C03639=1023.462,361.874,355.874,171.924,48.820,159.677
C03640=1023.470,362.121,355.836,171.932,48.821,159.679
C03641=1023.477,362.367,355.796,171.939,48.821,159.680
C03642=1023.485,362.615,355.758,171.947,48.820,159.681
C03643=1023.494,362.861,355.718,171.955,48.820,159.682
C03644=1023.502,363.108,355.680,171.963,48.820,159.683
C03645=1023.510,363.355,355.640,171.971,48.820,159.684
C03646=1023.517,363.602,355.602,171.978,48.820,159.685
C03647=1023.526,363.848,355.562,171.986,48.819,159.687
C03648=1023.534,364.095,355.523,171.994,48.820,159.688
C03649=1023.542,364.342,355.484,172.001,48.820,159.689
C03650=1023.551,364.589,355.445,172.009,48.819,159.690
C03651=1023.558,364.836,355.405,172.018,48.819,159.691
C03652=1023.567,365.083,355.366,172.025,48.819,159.692
C03653=1023.575,365.330,355.327,172.033,48.820,159.694
C03654=1023.583,365.576,355.288,172.041,48.819,159.695
C03655=1023.591,365.813,355.250,172.049,48.819,159.696
C03656=1023.599,366.049,355.212,172.057,48.819,159.697
C03657=1023.608,366.287,355.175,172.064,48.819,159.698
C03658=1023.615,366.524,355.137,172.072,48.819,159.700
C03659=1023.623,366.761,355.099,172.080,48.819,159.701
C03660=1023.631,366.998,355.060,172.088,48.820,159.702
C03661=1023.639,367.235,355.023,172.095,48.820,159.703
C03662=1023.647,367.471,354.985,172.103,48.819,159.704
C03663=1023.656,367.719,354.945,172.111,48.820,159.705
C03664=1023.664,367.965,354.906,172.119,48.820,159.707
C03665=1023.673,368.212,354.866,172.127,48.819,159.708
C03666=1023.680,368.459,354.826,172.135,48.820,159.709
C03667=1023.689,368.705,354.787,172.144,48.820,159.710
C03668=1023.697,368.952,354.747,172.151,48.820,159.712
C03669=1023.705,369.198,354.707,172.160,48.821,159.713
C03670=1023.713,369.445,354.667,172.168,48.821,159.714
C03671=1023.722,369.693,354.628,172.177,48.821,159.716
C03672=1023.730,369.939,354.587,172.185,48.821,159.717
C03673=1023.739,370.185,354.548,172.192,48.822,159.718
C03674=1023.747,370.432,354.507,172.201,48.822,159.719
C03675=1023.755,370.678,354.468,172.209,48.822,159.721
C03676=1023.764,370.925,354.427,172.218,48.822,159.722
C03677=1023.772,371.172,354.387,172.226,48.823,159.723
C03678=1023.780,371.418,354.347,172.235,48.823,159.725
C03679=1023.789,371.665,354.307,172.243,48.823,159.726
C03680=1023.797,371.912,354.266,172.250,48.824,159.727
C03681=1023.806,372.158,354.226,172.259,48.824,159.729
C03682=1023.814,372.405,354.186,172.267,48.824,159.730
C03683=1023.822,372.652,354.145,172.276,48.825,159.731
C03684=1023.831,372.898,354.105,172.284,48.825,159.733
C03685=1023.839,373.145,354.065,172.293,48.825,159.734
C03686=1023.848,373.391,354.025,172.301,48.825,159.735
C03687=1023.856,373.637,353.984,172.310,48.826,159.737
C03688=1023.866,373.884,353.944,172.319,48.826,159.738
C03689=1023.874,374.130,353.903,172.327,48.826,159.740
C03690=1023.883,374.377,353.863,172.336,48.827,159.741
C03691=1023.891,374.623,353.822,172.344,48.827,159.742
C03692=1023.900,374.870,353.782,172.353,48.828,159.744
C03693=1023.908,375.117,353.742,172.361,48.828,159.745
C03694=1023.917,375.364,353.702,172.370,48.829,159.747
C03695=1023.926,375.609,353.660,172.379,48.829,159.748
C03696=1023.935,375.856,353.620,172.387,48.830,159.750
C03697=1023.943,376.102,353.579,172.396,48.830,159.751
C03698=1023.952,376.349,353.538,172.405,48.831,159.752
C03699=1023.961,376.596,353.498,172.413,48.831,159.754
C03700=1023.969,376.842,353.457,172.422,48.832,159.755
C03701=1023.978,377.089,353.415,172.431,48.833,159.757
C03702=1023.987,377.336,353.374,172.439,48.833,159.758
C03703=1023.995,377.582,353.334,172.448,48.834,159.760
C03704=1024.004,377.828,353.293,172.457,48.835,159.761
C03705=1024.013,378.074,353.252,172.466,48.835,159.763
C03706=1024.021,378.320,353.210,172.475,48.836,159.764
C03707=1024.030,378.567,353.169,172.484,48.837,159.766
C03708=1024.038,378.813,353.128,172.493,48.838,159.767
C03709=1024.047,379.060,353.087,172.501,48.838,159.769
C03710=1024.056,379.306,353.045,172.510,48.839,159.770
C03711=1024.065,379.553,353.003,172.519,48.840,159.772
C03712=1024.073,379.799,352.963,172.528,48.841,159.773
C03713=1024.083,380.045,352.922,172.538,48.841,159.775
C03714=1024.092,380.292,352.880,172.546,48.842,159.776
C03715=1024.100,380.541,352.838,172.555,48.843,159.778
C03716=1024.109,380.790,352.797,172.564,48.843,159.779
C03717=1024.118,381.039,352.754,172.574,48.844,159.781
C03718=1024.127,381.288,352.713,172.583,48.845,159.783
C03719=1024.136,381.535,352.671,172.592,48.846,159.784
C03720=1024.145,381.781,352.629,172.601,48.846,159.786
C03721=1024.154,382.027,352.588,172.610,48.847,159.787
C03722=1024.163,382.274,352.546,172.619,48.849,159.789
C03723=1024.172,382.520,352.504,172.628,48.849,159.791
C03724=1024.181,382.766,352.463,172.638,48.850,159.792
C03725=1024.190,383.013,352.421,172.647,48.851,159.794
C03726=1024.199,383.259,352.380,172.656,48.852,159.795
C03727=1024.208,383.505,352.338,172.666,48.852,159.797
C03728=1024.217,383.752,352.296,172.675,48.854,159.799
C03729=1024.226,383.998,352.255,172.684,48.854,159.800
C03730=1024.235,384.244,352.212,172.694,48.855,159.802
C03731=1024.244,384.490,352.170,172.702,48.856,159.804
C03732=1024.253,384.737,352.129,172.713,48.857,159.805
C03733=1024.263,384.983,352.087,172.722,48.859,159.807
C03734=1024.273,385.229,352.045,172.730,48.859,159.809
C03735=1024.282,385.475,352.003,172.741,48.860,159.810
C03736=1024.290,385.722,351.961,172.749,48.861,159.812
C03737=1024.300,385.968,351.919,172.760,48.862,159.814
C03738=1024.309,386.215,351.877,172.769,48.863,159.816
C03739=1024.318,386.460,351.834,172.779,48.864,159.817
C03740=1024.327,386.706,351.791,172.788,48.866,159.819
C03741=1024.336,386.953,351.750,172.797,48.867,159.821
C03742=1024.346,387.199,351.707,172.807,48.868,159.822
C03743=1024.355,387.445,351.664,172.816,48.869,159.824
C03744=1024.364,387.691,351.623,172.826,48.870,159.826
C03745=1024.373,387.937,351.580,172.835,48.871,159.828
C03746=1024.383,388.183,351.537,172.845,48.872,159.829
C03747=1024.391,388.430,351.494,172.856,48.873,159.831
C03748=1024.401,388.676,351.452,172.865,48.875,159.833
C03749=1024.411,388.922,351.409,172.875,48.876,159.835
C03750=1024.420,389.167,351.367,172.884,48.877,159.837
C03751=1024.429,389.414,351.323,172.894,48.878,159.838
C03752=1024.438,389.660,351.281,172.904,48.880,159.840
C03753=1024.448,389.906,351.238,172.914,48.881,159.842
C03754=1024.457,390.152,351.196,172.924,48.882,159.844
C03755=1024.466,390.398,351.153,172.933,48.884,159.846
C03756=1024.476,390.645,351.110,172.944,48.885,159.848
C03757=1024.485,390.890,351.067,172.954,48.886,159.849
C03758=1024.494,391.137,351.023,172.963,48.888,159.851
C03759=1024.504,391.383,350.981,172.974,48.889,159.853
C03760=1024.513,391.629,350.938,172.984,48.890,159.855
C03761=1024.523,391.875,350.894,172.993,48.892,159.857
C03762=1024.532,392.121,350.852,173.003,48.893,159.859
C03763=1024.542,392.367,350.809,173.014,48.895,159.861
C03764=1024.551,392.613,350.765,173.023,48.897,159.863
C03765=1024.560,392.859,350.722,173.034,48.897,159.864
C03766=1024.571,393.105,350.679,173.044,48.899,159.866
C03767=1024.580,393.351,350.635,173.055,48.901,159.869
C03768=1024.589,393.597,350.592,173.065,48.902,159.870
C03769=1024.599,393.843,350.548,173.074,48.903,159.872
C03770=1024.609,394.089,350.505,173.085,48.905,159.874
C03771=1024.617,394.335,350.462,173.095,48.907,159.876
C03772=1024.627,394.580,350.418,173.106,48.908,159.878
C03773=1024.637,394.827,350.374,173.116,48.910,159.880
C03774=1024.647,395.072,350.330,173.126,48.912,159.882
C03775=1024.658,395.359,350.280,173.139,48.913,159.885
C03776=1024.669,395.643,350.229,173.150,48.915,159.887
C03777=1024.681,395.930,350.179,173.162,48.917,159.889
C03778=1024.692,396.216,350.127,173.174,48.919,159.892
C03779=1024.702,396.461,350.083,173.185,48.921,159.894
C03780=1024.711,396.708,350.039,173.195,48.922,159.896
C03781=1024.721,396.953,349.996,173.206,48.924,159.898
C03782=1024.731,397.199,349.952,173.216,48.925,159.900
C03783=1024.741,397.445,349.907,173.227,48.927,159.902
C03784=1024.751,397.691,349.863,173.238,48.929,159.904
C03785=1024.761,397.937,349.820,173.248,48.931,159.906
C03786=1024.770,398.183,349.776,173.259,48.933,159.908
C03787=1024.781,398.428,349.731,173.270,48.934,159.910
C03788=1024.790,398.674,349.687,173.281,48.936,159.912
C03789=1024.800,398.920,349.643,173.291,48.938,159.914
C03790=1024.810,399.165,349.599,173.302,48.940,159.917
C03791=1024.820,399.411,349.554,173.312,48.941,159.919
C03792=1024.830,399.658,349.510,173.324,48.943,159.921
C03793=1024.840,399.903,349.466,173.335,48.945,159.923
C03794=1024.850,400.149,349.421,173.346,48.947,159.925
C03795=1024.860,400.394,349.376,173.357,48.949,159.927
C03796=1024.869,400.640,349.332,173.367,48.951,159.929
C03797=1024.880,400.886,349.287,173.378,48.953,159.932
C03798=1024.890,401.132,349.242,173.389,48.955,159.934
C03799=1024.899,401.377,349.198,173.401,48.956,159.936
C03800=1024.909,401.623,349.153,173.411,48.959,159.938
C03801=1024.919,401.869,349.108,173.422,48.961,159.940
C03802=1024.929,402.114,349.063,173.433,48.963,159.943
C03803=1024.940,402.360,349.018,173.445,48.964,159.945
C03804=1024.950,402.606,348.973,173.456,48.967,159.947
C03805=1024.960,402.851,348.928,173.467,48.969,159.950
C03806=1024.970,403.097,348.883,173.478,48.971,159.952
C03807=1024.980,403.342,348.838,173.490,48.973,159.954
C03808=1024.990,403.588,348.793,173.501,48.975,159.956
C03809=1025.000,403.834,348.748,173.512,48.978,159.959
C03810=1025.010,404.079,348.702,173.524,48.980,159.961
C03811=1025.020,404.325,348.657,173.535,48.982,159.963
C03812=1025.030,404.571,348.612,173.547,48.984,159.966
C03813=1025.041,404.816,348.566,173.558,48.986,159.968
C03814=1025.051,405.063,348.521,173.569,48.988,159.970
C03815=1025.062,405.307,348.476,173.581,48.990,159.973
C03816=1025.072,405.553,348.431,173.592,48.992,159.975
C03817=1025.083,405.799,348.385,173.604,48.995,159.977
C03818=1025.093,406.044,348.339,173.615,48.997,159.980
C03819=1025.103,406.290,348.294,173.627,48.999,159.982
C03820=1025.114,406.536,348.248,173.638,49.002,159.985
C03821=1025.124,406.781,348.202,173.651,49.004,159.987
C03822=1025.134,407.026,348.157,173.662,49.006,159.989
C03823=1025.145,407.272,348.112,173.674,49.008,159.992
C03824=1025.155,407.518,348.066,173.686,49.011,159.994
C03825=1025.166,407.763,348.020,173.697,49.013,159.997
C03826=1025.176,408.009,347.974,173.709,49.016,159.999
C03827=1025.188,408.254,347.929,173.722,49.018,160.002
C03828=1025.198,408.500,347.883,173.733,49.020,160.004
C03829=1025.209,408.746,347.837,173.745,49.023,160.007
C03830=1025.220,408.991,347.791,173.757,49.025,160.009
C03831=1025.230,409.237,347.745,173.770,49.027,160.012
C03832=1025.241,409.482,347.699,173.781,49.030,160.014
C03833=1025.252,409.727,347.653,173.793,49.032,160.017
C03834=1025.263,409.973,347.607,173.806,49.035,160.019
C03835=1025.275,410.282,347.548,173.821,49.038,160.022
C03836=1025.289,410.590,347.489,173.836,49.041,160.026
C03837=1025.302,410.898,347.432,173.851,49.044,160.029
C03838=1025.316,411.206,347.373,173.867,49.048,160.032
C03839=1025.326,411.451,347.327,173.879,49.050,160.035
C03840=1025.337,411.697,347.279,173.891,49.053,160.037
C03841=1025.348,411.942,347.233,173.904,49.056,160.040
C03842=1025.359,412.188,347.187,173.916,49.058,160.043
C03843=1025.370,412.433,347.140,173.929,49.061,160.045
C03844=1025.380,412.679,347.093,173.941,49.063,160.048
C03845=1025.391,412.924,347.046,173.954,49.066,160.051
C03846=1025.402,413.169,346.999,173.966,49.068,160.053
C03847=1025.414,413.414,346.952,173.979,49.071,160.056
C03848=1025.424,413.660,346.905,173.992,49.074,160.059
C03849=1025.435,413.905,346.859,174.004,49.077,160.062
C03850=1025.446,414.150,346.812,174.017,49.080,160.064
C03851=1025.457,414.395,346.765,174.029,49.082,160.067
C03852=1025.468,414.641,346.717,174.042,49.085,160.070
C03853=1025.479,414.886,346.671,174.055,49.088,160.072
C03854=1025.491,415.131,346.623,174.069,49.091,160.075
C03855=1025.502,415.377,346.576,174.081,49.094,160.078
C03856=1025.513,415.622,346.529,174.094,49.097,160.081
C03857=1025.524,415.868,346.482,174.106,49.099,160.084
C03858=1025.535,416.113,346.434,174.119,49.103,160.087
C03859=1025.546,416.358,346.387,174.133,49.105,160.089
C03860=1025.557,416.604,346.339,174.146,49.108,160.092
C03861=1025.569,416.849,346.291,174.159,49.111,160.095
C03862=1025.579,417.094,346.244,174.173,49.114,160.098
C03863=1025.591,417.339,346.196,174.185,49.117,160.101
C03864=1025.602,417.584,346.148,174.198,49.120,160.104
C03865=1025.614,417.829,346.100,174.212,49.123,160.107
C03866=1025.625,418.074,346.052,174.225,49.127,160.110
C03867=1025.636,418.320,346.005,174.238,49.129,160.112
C03868=1025.647,418.565,345.957,174.252,49.132,160.115
C03869=1025.659,418.810,345.909,174.265,49.136,160.118
C03870=1025.670,419.056,345.861,174.279,49.139,160.121
C03871=1025.682,419.300,345.812,174.292,49.142,160.124
C03872=1025.693,419.545,345.764,174.306,49.145,160.127
C03873=1025.705,419.790,345.716,174.320,49.148,160.130
C03874=1025.716,420.036,345.668,174.333,49.151,160.133
C03875=1025.728,420.281,345.620,174.347,49.155,160.136
C03876=1025.740,420.526,345.571,174.360,49.158,160.139
C03877=1025.751,420.771,345.524,174.374,49.161,160.142
C03878=1025.762,421.016,345.475,174.388,49.164,160.145
C03879=1025.775,421.260,345.427,174.401,49.167,160.149
C03880=1025.786,421.506,345.379,174.415,49.170,160.152
C03881=1025.798,421.751,345.330,174.430,49.174,160.155
C03882=1025.810,421.996,345.282,174.444,49.177,160.158
C03883=1025.821,422.241,345.233,174.458,49.180,160.161
C03884=1025.833,422.485,345.184,174.471,49.184,160.164
C03885=1025.845,422.731,345.135,174.485,49.187,160.167
C03886=1025.857,422.976,345.086,174.500,49.190,160.170
C03887=1025.868,423.220,345.037,174.514,49.194,160.174
C03888=1025.881,423.466,344.988,174.528,49.197,160.177
C03889=1025.892,423.710,344.939,174.542,49.200,160.180
C03890=1025.903,423.955,344.890,174.557,49.204,160.183
C03891=1025.915,424.200,344.841,174.571,49.207,160.186
C03892=1025.928,424.445,344.792,174.585,49.211,160.190
C03893=1025.940,424.690,344.743,174.600,49.215,160.193
C03894=1025.951,424.935,344.694,174.615,49.218,160.196
C03895=1025.967,425.254,344.629,174.633,49.223,160.201
C03896=1025.982,425.573,344.565,174.652,49.227,160.205
C03897=1025.998,425.892,344.501,174.671,49.232,160.209
C03898=1026.014,426.211,344.437,174.691,49.236,160.214
C03899=1026.027,426.455,344.387,174.706,49.240,160.217
C03900=1026.039,426.701,344.337,174.720,49.244,160.220
C03901=1026.050,426.945,344.287,174.735,49.248,160.224
C03902=1026.063,427.190,344.237,174.750,49.251,160.227
C03903=1026.075,427.435,344.187,174.765,49.255,160.230
C03904=1026.087,427.679,344.137,174.780,49.259,160.234
C03905=1026.099,427.924,344.087,174.795,49.262,160.237
C03906=1026.111,428.168,344.037,174.810,49.266,160.241
C03907=1026.124,428.413,343.987,174.825,49.270,160.244
C03908=1026.136,428.658,343.937,174.840,49.274,160.248
C03909=1026.148,428.903,343.887,174.855,49.278,160.251
C03910=1026.160,429.148,343.837,174.871,49.281,160.255
C03911=1026.173,429.393,343.787,174.886,49.285,160.258
C03912=1026.185,429.637,343.736,174.901,49.289,160.262
C03913=1026.198,429.882,343.686,174.918,49.293,160.266
C03914=1026.210,430.126,343.635,174.932,49.297,160.269
C03915=1026.223,430.371,343.585,174.948,49.300,160.273
C03916=1026.235,430.615,343.535,174.963,49.305,160.276
C03917=1026.248,430.860,343.484,174.979,49.308,160.280
C03918=1026.261,431.105,343.433,174.995,49.312,160.284
C03919=1026.273,431.349,343.383,175.011,49.316,160.287
C03920=1026.286,431.594,343.332,175.027,49.320,160.291
C03921=1026.298,431.838,343.281,175.042,49.324,160.294
C03922=1026.312,432.083,343.230,175.058,49.329,160.298
C03923=1026.324,432.327,343.180,175.074,49.333,160.302
C03924=1026.337,432.572,343.129,175.090,49.337,160.306
C03925=1026.350,432.817,343.078,175.107,49.341,160.309
C03926=1026.363,433.061,343.027,175.123,49.345,160.313
C03927=1026.376,433.306,342.976,175.139,49.349,160.317
C03928=1026.389,433.550,342.924,175.155,49.353,160.321
C03929=1026.402,433.794,342.873,175.171,49.357,160.324
C03930=1026.414,434.038,342.822,175.188,49.361,160.328
C03931=1026.428,434.283,342.771,175.204,49.365,160.332
C03932=1026.441,434.528,342.719,175.220,49.370,160.336
C03933=1026.453,434.771,342.667,175.237,49.374,160.340
C03934=1026.466,435.016,342.616,175.254,49.378,160.344
C03935=1026.480,435.261,342.564,175.270,49.382,160.348
C03936=1026.493,435.505,342.513,175.287,49.387,160.352
C03937=1026.506,435.749,342.462,175.304,49.391,160.356
C03938=1026.519,435.994,342.409,175.321,49.396,160.360
C03939=1026.532,436.237,342.357,175.337,49.400,160.363
C03940=1026.545,436.482,342.306,175.354,49.404,160.367
C03941=1026.559,436.726,342.254,175.371,49.408,160.371
C03942=1026.572,436.970,342.201,175.389,49.413,160.376
C03943=1026.585,437.215,342.149,175.405,49.417,160.380
C03944=1026.599,437.459,342.097,175.423,49.422,160.384
C03945=1026.612,437.703,342.046,175.439,49.426,160.388
C03946=1026.625,437.947,341.992,175.457,49.431,160.392
C03947=1026.639,438.192,341.940,175.475,49.435,160.396
C03948=1026.652,438.436,341.889,175.491,49.439,160.400
C03949=1026.666,438.680,341.835,175.509,49.444,160.404
C03950=1026.679,438.924,341.783,175.527,49.449,160.409
C03951=1026.693,439.168,341.731,175.543,49.453,160.413
C03952=1026.706,439.412,341.678,175.561,49.458,160.417
C03953=1026.720,439.656,341.626,175.579,49.462,160.421
C03954=1026.734,439.900,341.573,175.597,49.467,160.425
C03955=1026.747,440.144,341.520,175.615,49.472,160.430
C03956=1026.760,440.390,341.467,175.633,49.476,160.434
C03957=1026.775,440.634,341.414,175.651,49.481,160.438
C03958=1026.789,440.879,341.360,175.669,49.486,160.442
C03959=1026.801,441.107,341.311,175.686,49.490,160.447
C03960=1026.815,441.334,341.262,175.703,49.495,160.451
C03961=1026.828,441.561,341.212,175.720,49.499,160.455
C03962=1026.840,441.790,341.162,175.736,49.503,160.459
C03963=1026.853,442.017,341.112,175.754,49.508,160.463
C03964=1026.867,442.244,341.063,175.771,49.512,160.467
C03965=1026.880,442.472,341.013,175.789,49.517,160.471
C03966=1026.893,442.700,340.964,175.805,49.521,160.475
C03967=1026.908,442.942,340.911,175.823,49.526,160.480
C03968=1026.922,443.185,340.858,175.842,49.530,160.484
C03969=1026.938,443.429,340.806,175.862,49.535,160.489
C03970=1026.954,443.673,340.755,175.879,49.540,160.493
C03971=1026.971,443.916,340.703,175.899,49.544,160.497
C03972=1026.987,444.160,340.653,175.918,49.548,160.502
C03973=1027.005,444.403,340.602,175.937,49.553,160.506
C03974=1027.022,444.648,340.552,175.956,49.557,160.511
C03975=1027.041,444.892,340.502,175.975,49.561,160.515
C03976=1027.060,445.136,340.453,175.994,49.565,160.519
C03977=1027.079,445.380,340.405,176.013,49.569,160.524
C03978=1027.098,445.624,340.356,176.033,49.573,160.528
C03979=1027.118,445.869,340.308,176.052,49.577,160.532
C03980=1027.138,446.113,340.261,176.072,49.581,160.537
C03981=1027.159,446.357,340.213,176.092,49.585,160.541
C03982=1027.181,446.601,340.166,176.112,49.588,160.545
C03983=1027.203,446.845,340.119,176.132,49.592,160.550
C03984=1027.225,447.091,340.073,176.151,49.596,160.554
C03985=1027.248,447.335,340.028,176.172,49.599,160.559
C03986=1027.272,447.580,339.983,176.192,49.603,160.563
C03987=1027.295,447.825,339.938,176.212,49.606,160.567
C03988=1027.319,448.069,339.893,176.232,49.609,160.571
C03989=1027.345,448.315,339.849,176.253,49.612,160.576
C03990=1027.369,448.559,339.805,176.274,49.615,160.580
C03991=1027.395,448.804,339.761,176.295,49.619,160.585
C03992=1027.421,449.049,339.719,176.315,49.621,160.589
C03993=1027.447,449.295,339.677,176.336,49.624,160.593
C03994=1027.475,449.539,339.635,176.357,49.628,160.597
C03995=1027.502,449.785,339.593,176.377,49.630,160.602
C03996=1027.530,450.030,339.551,176.399,49.633,160.606
C03997=1027.559,450.275,339.510,176.419,49.636,160.610
C03998=1027.587,450.521,339.469,176.441,49.638,160.615
C03999=1027.617,450.766,339.429,176.462,49.641,160.619
C04000=1027.646,451.012,339.389,176.483,49.644,160.623
C04001=1027.677,451.257,339.350,176.504,49.647,160.628
C04002=1027.707,451.502,339.311,176.526,49.649,160.632
C04003=1027.738,451.748,339.272,176.548,49.651,160.636
C04004=1027.771,451.994,339.235,176.570,49.653,160.640
C04005=1027.802,452.240,339.196,176.591,49.656,160.645
C04006=1027.835,452.485,339.159,176.614,49.658,160.649
C04007=1027.868,452.731,339.122,176.635,49.660,160.653
C04008=1027.902,452.977,339.086,176.658,49.662,160.658
C04009=1027.935,453.222,339.050,176.680,49.664,160.662
C04010=1027.971,453.468,339.013,176.703,49.666,160.666
C04011=1028.005,453.714,338.979,176.725,49.668,160.671
C04012=1028.040,453.960,338.943,176.747,49.670,160.675
C04013=1028.076,454.206,338.909,176.770,49.672,160.679
C04014=1028.113,454.451,338.875,176.792,49.674,160.683
C04015=1027.838,454.527,338.537,176.795,49.734,160.703
C04016=1027.801,454.282,338.572,176.773,49.732,160.699
C04017=1027.765,454.036,338.606,176.749,49.731,160.694
C04018=1027.730,453.790,338.641,176.727,49.729,160.690
C04019=1027.695,453.544,338.676,176.705,49.727,160.686
C04020=1027.660,453.298,338.711,176.682,49.725,160.681
C04021=1027.626,453.053,338.748,176.660,49.723,160.677
C04022=1027.593,452.807,338.785,176.638,49.722,160.673
C04023=1027.560,452.561,338.821,176.616,49.719,160.669
C04024=1027.527,452.316,338.858,176.594,49.717,160.664
C04025=1027.494,452.070,338.896,176.572,49.715,160.660
C04026=1027.463,451.824,338.934,176.550,49.713,160.656
C04027=1027.431,451.578,338.972,176.528,49.711,160.652
C04028=1027.400,451.334,339.012,176.506,49.708,160.647
C04029=1027.370,451.088,339.050,176.485,49.706,160.643
C04030=1027.340,450.842,339.090,176.463,49.703,160.639
C04031=1027.310,450.596,339.130,176.442,49.701,160.634
C04032=1027.281,450.351,339.171,176.421,49.699,160.630
C04033=1027.253,450.106,339.211,176.400,49.695,160.626
C04034=1027.224,449.861,339.252,176.378,49.693,160.621
C04035=1027.197,449.616,339.294,176.358,49.690,160.617
C04036=1027.170,449.370,339.336,176.336,49.687,160.613
C04037=1027.143,449.126,339.378,176.316,49.685,160.609
C04038=1027.117,448.880,339.421,176.295,49.681,160.604
C04039=1027.091,448.635,339.465,176.274,49.679,160.600
C04040=1027.065,448.390,339.508,176.254,49.676,160.596
C04041=1027.041,448.145,339.551,176.233,49.672,160.591
C04042=1027.016,447.900,339.596,176.213,49.670,160.587
C04043=1026.992,447.656,339.641,176.193,49.666,160.583
C04044=1026.969,447.411,339.686,176.172,49.663,160.578
C04045=1026.945,447.166,339.732,176.152,49.659,160.574
C04046=1026.923,446.921,339.777,176.132,49.656,160.570
C04047=1026.902,446.677,339.824,176.112,49.653,160.565
C04048=1026.880,446.432,339.871,176.092,49.649,160.561
C04049=1026.858,446.187,339.918,176.072,49.646,160.557
C04050=1026.838,445.944,339.965,176.052,49.642,160.552
C04051=1026.817,445.699,340.013,176.033,49.638,160.548
C04052=1026.798,445.455,340.061,176.013,49.634,160.544
C04053=1026.778,445.210,340.110,175.994,49.630,160.539
C04054=1026.759,444.967,340.159,175.975,49.626,160.535
C04055=1026.741,444.723,340.209,175.956,49.622,160.531
C04056=1026.723,444.479,340.258,175.936,49.618,160.526
C04057=1026.705,444.234,340.308,175.917,49.614,160.522
C04058=1026.688,443.991,340.359,175.898,49.610,160.517
C04059=1026.671,443.748,340.410,175.879,49.606,160.513
C04060=1026.655,443.503,340.461,175.860,49.601,160.508
C04061=1026.639,443.260,340.514,175.842,49.597,160.504
C04062=1026.625,443.017,340.566,175.823,49.592,160.500
C04063=1026.610,442.774,340.619,175.804,49.587,160.495
C04064=1026.595,442.531,340.671,175.786,49.583,160.491
C04065=1026.581,442.287,340.725,175.767,49.578,160.486
C04066=1026.567,442.043,340.777,175.749,49.573,160.482
C04067=1026.553,441.800,340.831,175.730,49.569,160.478
C04068=1026.540,441.576,340.879,175.714,49.565,160.474
C04069=1026.527,441.353,340.928,175.697,49.561,160.470
C04070=1026.515,441.129,340.976,175.681,49.556,160.466
C04071=1026.502,440.905,341.025,175.664,49.552,160.462
C04072=1026.489,440.681,341.074,175.648,49.547,160.458
C04073=1026.477,440.458,341.123,175.630,49.544,160.454
C04074=1026.464,440.234,341.171,175.614,49.540,160.450
C04075=1026.452,440.011,341.219,175.597,49.535,160.446
C04076=1026.438,439.766,341.273,175.580,49.531,160.442
C04077=1026.424,439.522,341.325,175.563,49.526,160.438
C04078=1026.411,439.278,341.377,175.545,49.521,160.433
C04079=1026.397,439.034,341.430,175.527,49.517,160.429
C04080=1026.384,438.790,341.483,175.509,49.513,160.425
C04081=1026.370,438.546,341.535,175.492,49.508,160.421
C04082=1026.357,438.302,341.588,175.474,49.504,160.417
C04083=1026.343,438.057,341.640,175.457,49.499,160.413
C04084=1026.329,437.813,341.692,175.440,49.495,160.408
C04085=1026.316,437.569,341.744,175.422,49.491,160.404
C04086=1026.303,437.325,341.797,175.405,49.486,160.400
C04087=1026.290,437.081,341.849,175.388,49.482,160.396
C04088=1026.276,436.837,341.901,175.371,49.478,160.392
C04089=1026.263,436.592,341.953,175.354,49.473,160.388
C04090=1026.249,436.348,342.004,175.337,49.469,160.384
C04091=1026.236,436.104,342.057,175.320,49.465,160.380
C04092=1026.219,435.783,342.125,175.298,49.459,160.375
C04093=1026.202,435.462,342.193,175.276,49.454,160.370
C04094=1026.184,435.142,342.260,175.254,49.449,160.365
C04095=1026.168,434.821,342.327,175.233,49.443,160.360
C04096=1026.154,434.577,342.379,175.215,49.439,160.356
C04097=1026.142,434.332,342.431,175.199,49.435,160.352
C04098=1026.129,434.088,342.483,175.183,49.431,160.348
C04099=1026.116,433.843,342.534,175.166,49.426,160.344
C04100=1026.103,433.599,342.585,175.150,49.422,160.340
C04101=1026.089,433.355,342.636,175.134,49.418,160.337
C04102=1026.077,433.111,342.687,175.117,49.414,160.333
C04103=1026.064,432.866,342.738,175.101,49.410,160.329
C04104=1026.051,432.621,342.789,175.085,49.406,160.325
C04105=1026.038,432.377,342.840,175.069,49.402,160.322
C04106=1026.025,432.132,342.891,175.053,49.399,160.318
C04107=1026.013,431.888,342.941,175.038,49.394,160.314
C04108=1026.000,431.643,342.992,175.021,49.390,160.311
C04109=1025.988,431.399,343.043,175.006,49.387,160.307
C04110=1025.974,431.154,343.094,174.990,49.383,160.303
C04111=1025.962,430.909,343.144,174.974,49.379,160.300
C04112=1025.949,430.665,343.195,174.958,49.375,160.296
C04113=1025.937,430.420,343.245,174.943,49.371,160.292
C04114=1025.924,430.176,343.296,174.927,49.368,160.289
C04115=1025.912,429.931,343.346,174.911,49.364,160.285
C04116=1025.900,429.687,343.396,174.896,49.360,160.282
C04117=1025.887,429.442,343.447,174.880,49.356,160.278
C04118=1025.875,429.198,343.497,174.865,49.353,160.275
C04119=1025.863,428.953,343.547,174.850,49.349,160.271
C04120=1025.850,428.708,343.597,174.834,49.345,160.268
C04121=1025.837,428.464,343.647,174.819,49.341,160.264
C04122=1025.825,428.219,343.698,174.804,49.338,160.261
C04123=1025.812,427.974,343.748,174.789,49.334,160.257
C04124=1025.800,427.730,343.798,174.773,49.330,160.254
C04125=1025.788,427.484,343.847,174.759,49.327,160.250
C04126=1025.776,427.240,343.897,174.743,49.323,160.247
C04127=1025.764,426.995,343.947,174.729,49.320,160.244
C04128=1025.752,426.750,343.997,174.714,49.316,160.240
C04129=1025.740,426.506,344.047,174.699,49.312,160.237
C04130=1025.728,426.261,344.096,174.684,49.309,160.233
C04131=1025.716,426.016,344.146,174.669,49.305,160.230
C04132=1025.704,425.770,344.196,174.654,49.302,160.227
C04133=1025.692,425.526,344.245,174.640,49.298,160.223
C04134=1025.679,425.281,344.294,174.625,49.295,160.220
C04135=1025.667,425.036,344.344,174.610,49.292,160.217
C04136=1025.656,424.791,344.393,174.596,49.288,160.214
C04137=1025.643,424.546,344.443,174.582,49.285,160.210
C04138=1025.631,424.302,344.491,174.567,49.281,160.207
C04139=1025.619,424.056,344.540,174.553,49.278,160.204
C04140=1025.608,423.812,344.589,174.538,49.274,160.201
C04141=1025.596,423.567,344.638,174.524,49.271,160.197
C04142=1025.584,423.322,344.687,174.510,49.268,160.194
C04143=1025.572,423.077,344.736,174.496,49.265,160.191
C04144=1025.561,422.832,344.785,174.481,49.261,160.188
C04145=1025.548,422.587,344.834,174.467,49.258,160.185
C04146=1025.537,422.342,344.882,174.453,49.255,160.182
C04147=1025.526,422.097,344.931,174.439,49.251,160.178
C04148=1025.514,421.852,344.980,174.425,49.249,160.175
C04149=1025.502,421.607,345.028,174.411,49.245,160.172
C04150=1025.490,421.362,345.077,174.397,49.242,160.169
C04151=1025.479,421.117,345.125,174.383,49.239,160.166
C04152=1025.467,420.872,345.174,174.369,49.235,160.163
C04153=1025.455,420.626,345.222,174.356,49.232,160.160
C04154=1025.444,420.381,345.271,174.342,49.229,160.157
C04155=1025.431,420.136,345.319,174.328,49.226,160.154
C04156=1025.420,419.891,345.367,174.314,49.223,160.151
C04157=1025.409,419.646,345.415,174.301,49.220,160.148
C04158=1025.397,419.401,345.463,174.287,49.217,160.145
C04159=1025.386,419.156,345.511,174.274,49.214,160.142
C04160=1025.375,418.910,345.559,174.260,49.211,160.139
C04161=1025.363,418.666,345.607,174.246,49.208,160.136
C04162=1025.352,418.421,345.655,174.233,49.205,160.133
C04163=1025.340,418.175,345.703,174.219,49.202,160.130
C04164=1025.329,417.930,345.751,174.206,49.199,160.127
C04165=1025.317,417.685,345.799,174.193,49.196,160.124
C04166=1025.306,417.440,345.847,174.179,49.193,160.121
C04167=1025.295,417.195,345.894,174.166,49.190,160.118
C04168=1025.284,416.949,345.942,174.153,49.188,160.116
C04169=1025.272,416.704,345.990,174.140,49.184,160.113
C04170=1025.262,416.459,346.037,174.127,49.182,160.110
C04171=1025.250,416.214,346.084,174.114,49.179,160.107
C04172=1025.239,415.969,346.133,174.101,49.176,160.104
C04173=1025.228,415.724,346.179,174.088,49.173,160.101
C04174=1025.218,415.478,346.227,174.074,49.171,160.099
C04175=1025.206,415.233,346.275,174.062,49.168,160.096
C04176=1025.195,414.988,346.321,174.049,49.165,160.093
C04177=1025.183,414.742,346.368,174.036,49.162,160.090
C04178=1025.173,414.497,346.415,174.023,49.160,160.088
C04179=1025.162,414.251,346.462,174.010,49.157,160.085
C04180=1025.151,414.006,346.509,173.998,49.154,160.082
C04181=1025.139,413.760,346.556,173.985,49.152,160.079
C04182=1025.129,413.515,346.603,173.972,49.149,160.077
C04183=1025.117,413.269,346.650,173.960,49.146,160.074
C04184=1025.106,413.024,346.697,173.947,49.144,160.071
C04185=1025.096,412.779,346.744,173.935,49.141,160.069
C04186=1025.085,412.533,346.791,173.922,49.138,160.066
C04187=1025.074,412.288,346.838,173.910,49.136,160.063
C04188=1025.063,412.043,346.884,173.897,49.133,160.061
C04189=1025.052,411.798,346.930,173.885,49.130,160.058
C04190=1025.042,411.553,346.977,173.872,49.128,160.055
C04191=1025.031,411.307,347.024,173.860,49.125,160.053
C04192=1025.018,410.997,347.083,173.844,49.123,160.050
C04193=1025.004,410.686,347.141,173.829,49.120,160.046
C04194=1024.990,410.375,347.201,173.813,49.116,160.043
C04195=1024.977,410.065,347.259,173.798,49.113,160.040
C04196=1024.966,409.820,347.306,173.786,49.111,160.037
C04197=1024.955,409.575,347.352,173.773,49.109,160.035
C04198=1024.945,409.329,347.397,173.761,49.106,160.032
C04199=1024.934,409.083,347.443,173.750,49.104,160.030
C04200=1024.924,408.838,347.489,173.738,49.101,160.027
C04201=1024.913,408.592,347.535,173.725,49.099,160.025
C04202=1024.902,408.347,347.581,173.713,49.097,160.022
C04203=1024.892,408.101,347.627,173.701,49.095,160.020
C04204=1024.881,407.855,347.673,173.690,49.092,160.017
C04205=1024.870,407.610,347.719,173.677,49.090,160.015
C04206=1024.860,407.364,347.765,173.666,49.088,160.012
C04207=1024.849,407.119,347.811,173.654,49.085,160.010
C04208=1024.839,406.873,347.856,173.642,49.083,160.007
C04209=1024.828,406.628,347.901,173.630,49.081,160.005
C04210=1024.817,406.382,347.947,173.619,49.079,160.003
C04211=1024.807,406.137,347.993,173.607,49.077,160.000
C04212=1024.797,405.890,348.038,173.596,49.075,159.998
C04213=1024.787,405.645,348.083,173.584,49.073,159.996
C04214=1024.776,405.400,348.129,173.573,49.070,159.993
C04215=1024.766,405.154,348.174,173.561,49.068,159.991
C04216=1024.756,404.909,348.220,173.549,49.066,159.988
C04217=1024.745,404.663,348.265,173.538,49.064,159.986
C04218=1024.736,404.417,348.310,173.527,49.062,159.984
C04219=1024.725,404.171,348.356,173.514,49.060,159.981
C04220=1024.714,403.926,348.400,173.504,49.058,159.979
C04221=1024.704,403.680,348.445,173.492,49.056,159.977
C04222=1024.694,403.435,348.491,173.481,49.054,159.975
C04223=1024.684,403.189,348.536,173.470,49.052,159.972
C04224=1024.674,402.943,348.581,173.458,49.050,159.970
C04225=1024.664,402.697,348.626,173.447,49.048,159.968
C04226=1024.654,402.452,348.672,173.436,49.046,159.966
C04227=1024.644,402.207,348.716,173.424,49.044,159.963
C04228=1024.634,401.961,348.762,173.414,49.042,159.961
C04229=1024.624,401.715,348.806,173.403,49.040,159.959
C04230=1024.614,401.470,348.851,173.391,49.038,159.957
C04231=1024.604,401.224,348.895,173.380,49.036,159.954
C04232=1024.594,400.978,348.940,173.369,49.034,159.952
C04233=1024.584,400.732,348.985,173.358,49.032,159.950
C04234=1024.574,400.487,349.029,173.347,49.031,159.948
C04235=1024.564,400.241,349.074,173.336,49.029,159.946
C04236=1024.554,399.994,349.118,173.325,49.027,159.944
C04237=1024.544,399.749,349.163,173.314,49.025,159.941
C04238=1024.534,399.504,349.207,173.303,49.023,159.939
C04239=1024.524,399.258,349.251,173.292,49.022,159.937
C04240=1024.515,399.012,349.296,173.281,49.020,159.935
C04241=1024.504,398.766,349.340,173.271,49.018,159.933
C04242=1024.495,398.521,349.385,173.260,49.017,159.931
C04243=1024.485,398.275,349.428,173.249,49.015,159.929
C04244=1024.474,398.029,349.473,173.239,49.013,159.927
C04245=1024.465,397.783,349.517,173.228,49.012,159.924
C04246=1024.455,397.537,349.561,173.217,49.010,159.922
C04247=1024.445,397.291,349.605,173.207,49.008,159.920
C04248=1024.435,397.045,349.648,173.196,49.006,159.918
C04249=1024.425,396.799,349.693,173.186,49.005,159.916
C04250=1024.415,396.553,349.737,173.175,49.003,159.914
C04251=1024.407,396.308,349.781,173.165,49.002,159.912
C04252=1024.395,396.019,349.832,173.151,49.000,159.910
C04253=1024.383,395.732,349.883,173.140,48.998,159.907
C04254=1024.372,395.444,349.934,173.127,48.997,159.905
C04255=1024.361,395.155,349.985,173.115,48.995,159.903
C04256=1024.351,394.909,350.029,173.104,48.993,159.901
C04257=1024.341,394.663,350.073,173.094,48.992,159.899
C04258=1024.332,394.418,350.116,173.083,48.990,159.897
C04259=1024.322,394.172,350.160,173.074,48.989,159.895
C04260=1024.312,393.925,350.203,173.064,48.987,159.893
C04261=1024.303,393.679,350.247,173.053,48.986,159.891
C04262=1024.294,393.434,350.290,173.043,48.984,159.889
C04263=1024.284,393.187,350.334,173.032,48.983,159.887
C04264=1024.274,392.942,350.377,173.022,48.982,159.885
C04265=1024.265,392.696,350.419,173.013,48.980,159.883
C04266=1024.256,392.450,350.464,173.002,48.979,159.881
C04267=1024.246,392.203,350.506,172.992,48.978,159.879
C04268=1024.236,391.958,350.550,172.982,48.976,159.877
C04269=1024.227,391.711,350.593,172.972,48.975,159.876
C04270=1024.218,391.466,350.635,172.962,48.973,159.874
C04271=1024.208,391.220,350.679,172.952,48.972,159.872
C04272=1024.199,390.973,350.722,172.942,48.971,159.870
C04273=1024.189,390.727,350.765,172.931,48.970,159.868
C04274=1024.180,390.481,350.808,172.922,48.969,159.866
C04275=1024.170,390.235,350.850,172.912,48.968,159.865
C04276=1024.162,389.990,350.894,172.901,48.966,159.863
C04277=1024.152,389.743,350.936,172.892,48.965,159.861
C04278=1024.142,389.498,350.979,172.882,48.964,159.859
C04279=1024.133,389.251,351.022,172.872,48.963,159.857
C04280=1024.124,389.005,351.065,172.863,48.961,159.855
C04281=1024.115,388.759,351.107,172.853,48.960,159.854
C04282=1024.105,388.513,351.150,172.843,48.959,159.852
C04283=1024.096,388.266,351.192,172.833,48.958,159.850
C04284=1024.087,388.020,351.235,172.823,48.957,159.848
C04285=1024.078,387.774,351.278,172.814,48.956,159.847
C04286=1024.069,387.528,351.320,172.804,48.955,159.845
C04287=1024.060,387.282,351.362,172.795,48.953,159.843
C04288=1024.050,387.035,351.404,172.785,48.953,159.841
C04289=1024.040,386.790,351.447,172.776,48.952,159.840
C04290=1024.032,386.543,351.489,172.766,48.951,159.838
C04291=1024.023,386.297,351.532,172.756,48.949,159.836
C04292=1024.014,386.050,351.574,172.746,48.948,159.834
C04293=1024.004,385.804,351.616,172.738,48.948,159.833
C04294=1023.995,385.558,351.658,172.727,48.947,159.831
C04295=1023.986,385.312,351.700,172.719,48.946,159.829
C04296=1023.977,385.066,351.742,172.708,48.945,159.828
C04297=1023.967,384.819,351.783,172.700,48.944,159.826
C04298=1023.958,384.573,351.825,172.690,48.943,159.824
C04299=1023.949,384.327,351.868,172.681,48.942,159.823
C04300=1023.940,384.081,351.909,172.671,48.941,159.821
C04301=1023.931,383.834,351.951,172.662,48.941,159.819
C04302=1023.922,383.588,351.993,172.653,48.939,159.818
C04303=1023.913,383.342,352.035,172.643,48.939,159.816
C04304=1023.904,383.095,352.076,172.634,48.938,159.815
C04305=1023.894,382.849,352.117,172.624,48.937,159.813
C04306=1023.885,382.603,352.159,172.615,48.936,159.811
C04307=1023.877,382.357,352.201,172.606,48.936,159.810
C04308=1023.868,382.110,352.242,172.597,48.935,159.808
C04309=1023.859,381.864,352.284,172.588,48.935,159.807
C04310=1023.850,381.617,352.326,172.579,48.933,159.805
C04311=1023.841,381.371,352.368,172.569,48.933,159.803
C04312=1023.832,381.119,352.410,172.560,48.932,159.802
C04313=1023.822,380.869,352.452,172.550,48.932,159.800
C04314=1023.814,380.618,352.494,172.541,48.931,159.799
C04315=1023.805,380.366,352.536,172.533,48.930,159.797
C04316=1023.796,380.119,352.578,172.523,48.930,159.795
C04317=1023.787,379.873,352.620,172.514,48.929,159.794
C04318=1023.779,379.627,352.660,172.505,48.928,159.792
C04319=1023.770,379.380,352.702,172.496,48.927,159.791
C04320=1023.760,379.134,352.743,172.488,48.927,159.789
C04321=1023.752,378.887,352.784,172.478,48.926,159.788
C04322=1023.743,378.642,352.826,172.469,48.925,159.786
C04323=1023.735,378.395,352.867,172.460,48.925,159.785
C04324=1023.726,378.148,352.908,172.452,48.924,159.783
C04325=1023.718,377.902,352.949,172.443,48.924,159.782
C04326=1023.709,377.656,352.991,172.434,48.923,159.780
C04327=1023.700,377.409,353.032,172.425,48.922,159.779
C04328=1023.691,377.163,353.072,172.416,48.922,159.777
C04329=1023.682,376.916,353.113,172.407,48.921,159.776
C04330=1023.674,376.670,353.154,172.398,48.921,159.774
C04331=1023.666,376.423,353.195,172.390,48.921,159.773
C04332=1023.656,376.176,353.235,172.381,48.920,159.772
C04333=1023.648,375.930,353.276,172.373,48.920,159.770
C04334=1023.639,375.684,353.317,172.364,48.919,159.769
C04335=1023.631,375.438,353.358,172.355,48.919,159.767
C04336=1023.621,375.191,353.398,172.346,48.919,159.766
C04337=1023.613,374.945,353.439,172.337,48.918,159.764
C04338=1023.605,374.697,353.479,172.329,48.918,159.763
C04339=1023.596,374.451,353.519,172.321,48.918,159.762
C04340=1023.587,374.204,353.560,172.312,48.917,159.760
C04341=1023.579,373.958,353.600,172.303,48.917,159.759
C04342=1023.570,373.711,353.641,172.295,48.916,159.758
C04343=1023.561,373.465,353.681,172.286,48.916,159.756
C04344=1023.553,373.219,353.722,172.278,48.916,159.755
C04345=1023.544,372.972,353.762,172.269,48.915,159.753
C04346=1023.536,372.726,353.802,172.261,48.915,159.752
C04347=1023.527,372.479,353.843,172.252,48.915,159.751
C04348=1023.519,372.232,353.883,172.244,48.915,159.749
C04349=1023.510,371.986,353.923,172.235,48.915,159.748
C04350=1023.502,371.739,353.964,172.227,48.914,159.747
C04351=1023.493,371.492,354.003,172.219,48.914,159.745
C04352=1023.485,371.246,354.044,172.210,48.914,159.744
C04353=1023.477,371.000,354.083,172.202,48.914,159.743
C04354=1023.468,370.753,354.124,172.194,48.913,159.742
C04355=1023.460,370.506,354.164,172.186,48.913,159.740
C04356=1023.452,370.260,354.204,172.177,48.913,159.739
C04357=1023.444,370.013,354.244,172.169,48.913,159.738
C04358=1023.435,369.767,354.284,172.161,48.913,159.736
C04359=1023.427,369.519,354.324,172.152,48.912,159.735
C04360=1023.418,369.273,354.363,172.144,48.912,159.734
C04361=1023.410,369.026,354.404,172.136,48.913,159.733
C04362=1023.402,368.780,354.443,172.128,48.912,159.731
C04363=1023.394,368.533,354.483,172.120,48.912,159.730
C04364=1023.386,368.286,354.523,172.111,48.912,159.729
C04365=1023.377,368.040,354.562,172.103,48.912,159.728
C04366=1023.370,367.793,354.602,172.095,48.912,159.726
C04367=1023.361,367.545,354.642,172.087,48.912,159.725
C04368=1023.353,367.308,354.680,172.079,48.912,159.724
C04369=1023.344,367.070,354.717,172.071,48.912,159.723
C04370=1023.336,366.832,354.755,172.064,48.912,159.721
C04371=1023.328,366.594,354.794,172.056,48.912,159.720
C04372=1023.320,366.355,354.832,172.048,48.912,159.719
C04373=1023.312,366.117,354.870,172.040,48.912,159.718
C04374=1023.305,365.879,354.908,172.032,48.912,159.717
C04375=1023.297,365.641,354.945,172.025,48.912,159.716
C04376=1023.288,365.394,354.985,172.017,48.912,159.714
C04377=1023.280,365.148,355.024,172.008,48.913,159.713
C04378=1023.272,364.901,355.063,172.001,48.913,159.712
C04379=1023.263,364.654,355.102,171.993,48.913,159.711
C04380=1023.256,364.407,355.142,171.985,48.913,159.710
C04381=1023.247,364.160,355.181,171.977,48.913,159.709
C04382=1023.239,363.913,355.220,171.970,48.913,159.708
C04383=1023.231,363.667,355.259,171.961,48.913,159.706
C04384=1023.223,363.421,355.298,171.953,48.914,159.705
C04385=1023.215,363.174,355.337,171.946,48.914,159.704
C04386=1023.207,362.927,355.377,171.938,48.914,159.703
C04387=1023.199,362.679,355.415,171.930,48.914,159.702
C04388=1023.190,362.433,355.455,171.923,48.915,159.701
C04389=1023.183,362.186,355.493,171.915,48.915,159.700
C04390=1023.174,361.940,355.532,171.906,48.915,159.698
C04391=1023.167,361.692,355.571,171.899,48.915,159.697
C04392=1023.159,361.445,355.610,171.891,48.915,159.696
C04393=1023.151,361.199,355.649,171.883,48.916,159.695
C04394=1023.143,360.952,355.688,171.876,48.916,159.694
C04395=1023.134,360.705,355.727,171.868,48.916,159.693
C04396=1023.127,360.459,355.765,171.861,48.916,159.692
C04397=1023.119,360.211,355.804,171.853,48.917,159.691
C04398=1023.111,359.964,355.843,171.845,48.918,159.690
C04399=1023.104,359.718,355.881,171.838,48.918,159.689
C04400=1023.095,359.470,355.920,171.830,48.918,159.688
C04401=1023.086,359.224,355.959,171.823,48.918,159.687
C04402=1023.079,358.978,355.997,171.815,48.919,159.686
C04403=1023.070,358.730,356.035,171.807,48.919,159.685
C04404=1023.063,358.484,356.074,171.800,48.920,159.684
C04405=1023.055,358.237,356.112,171.792,48.920,159.682
C04406=1023.047,357.989,356.151,171.785,48.921,159.682
C04407=1023.039,357.742,356.188,171.777,48.921,159.680
C04408=1023.031,357.495,356.227,171.770,48.921,159.679
C04409=1023.024,357.248,356.265,171.762,48.922,159.678
C04410=1023.015,357.002,356.303,171.754,48.922,159.677
C04411=1023.007,356.755,356.341,171.747,48.923,159.676
C04412=1022.999,356.508,356.380,171.739,48.924,159.675
C04413=1022.992,356.261,356.418,171.733,48.924,159.674
C04414=1022.984,356.014,356.456,171.725,48.925,159.673
C04415=1022.976,355.767,356.494,171.718,48.925,159.673
C04416=1022.968,355.519,356.532,171.710,48.926,159.671
C04417=1022.960,355.273,356.570,171.703,48.926,159.671
C04418=1022.952,355.026,356.608,171.695,48.927,159.669
C04419=1022.945,354.779,356.646,171.688,48.927,159.669
C04420=1022.937,354.532,356.684,171.680,48.928,159.668
C04421=1022.930,354.285,356.722,171.673,48.928,159.667
C04422=1022.921,354.038,356.760,171.666,48.929,159.666
C04423=1022.914,353.791,356.797,171.659,48.930,159.665
C04424=1022.906,353.544,356.836,171.652,48.931,159.664
C04425=1022.898,353.297,356.873,171.644,48.931,159.663
C04426=1022.890,353.050,356.910,171.637,48.932,159.662
C04427=1022.882,352.803,356.949,171.630,48.933,159.661
C04428=1022.875,352.568,356.984,171.623,48.934,159.660
C04429=1022.867,352.333,357.020,171.616,48.934,159.659
C04430=1022.860,352.099,357.056,171.609,48.935,159.658
C04431=1022.852,351.864,357.091,171.603,48.936,159.658
C04432=1022.845,351.630,357.127,171.596,48.936,159.657
C04433=1022.838,351.395,357.163,171.589,48.937,159.656
C04434=1022.831,351.160,357.199,171.582,48.938,159.655
C04435=1022.823,350.925,357.234,171.575,48.939,159.654
C04436=1022.816,350.678,357.272,171.568,48.939,159.653
C04437=1022.808,350.431,357.309,171.561,48.940,159.652
C04438=1022.801,350.185,357.347,171.554,48.941,159.652
C04439=1022.793,349.938,357.384,171.547,48.942,159.651
C04440=1022.785,349.690,357.422,171.539,48.943,159.650
C04441=1022.778,349.443,357.459,171.532,48.943,159.649
C04442=1022.770,349.196,357.496,171.526,48.944,159.648
C04443=1022.762,348.949,357.534,171.518,48.945,159.647
C04444=1022.755,348.702,357.571,171.512,48.946,159.646
C04445=1022.747,348.455,357.608,171.505,48.947,159.646
C04446=1022.740,348.208,357.646,171.497,48.948,159.645
C04447=1022.732,347.960,357.682,171.490,48.949,159.644
C04448=1022.725,347.713,357.719,171.484,48.949,159.643
C04449=1022.717,347.466,357.756,171.476,48.951,159.642
C04450=1022.710,347.219,357.794,171.470,48.951,159.641
C04451=1022.702,346.972,357.831,171.463,48.952,159.641
C04452=1022.695,346.725,357.868,171.455,48.954,159.640
C04453=1022.687,346.478,357.905,171.449,48.954,159.639
C04454=1022.679,346.231,357.942,171.442,48.955,159.638
C04455=1022.672,345.983,357.978,171.435,48.957,159.637
C04456=1022.664,345.736,358.015,171.428,48.957,159.637
C04457=1022.656,345.489,358.052,171.421,48.959,159.636
C04458=1022.649,345.242,358.089,171.415,48.959,159.635
C04459=1022.641,344.994,358.125,171.407,48.960,159.634
C04460=1022.634,344.747,358.163,171.401,48.962,159.633
C04461=1022.626,344.500,358.200,171.394,48.962,159.633
C04462=1022.618,344.253,358.236,171.386,48.964,159.632
C04463=1022.612,344.005,358.273,171.380,48.965,159.631
C04464=1022.604,343.758,358.310,171.373,48.966,159.630
C04465=1022.596,343.511,358.346,171.367,48.967,159.630
C04466=1022.589,343.265,358.383,171.359,48.968,159.629
C04467=1022.582,343.017,358.419,171.353,48.969,159.628
C04468=1022.574,342.770,358.455,171.346,48.971,159.627
C04469=1022.567,342.523,358.493,171.340,48.971,159.627
C04470=1022.559,342.275,358.529,171.332,48.973,159.626
C04471=1022.551,342.028,358.565,171.326,48.974,159.625
C04472=1022.545,341.781,358.602,171.319,48.975,159.624
C04473=1022.537,341.534,358.639,171.313,48.976,159.624
C04474=1022.529,341.286,358.675,171.306,48.978,159.623
C04475=1022.522,341.039,358.711,171.299,48.979,159.622
C04476=1022.515,340.792,358.748,171.292,48.980,159.621
C04477=1022.508,340.544,358.784,171.286,48.981,159.621
C04478=1022.500,340.297,358.820,171.280,48.982,159.620
C04479=1022.494,340.050,358.857,171.273,48.984,159.619
C04480=1022.486,339.802,358.893,171.266,48.985,159.619
C04481=1022.478,339.556,358.930,171.259,48.987,159.618
C04482=1022.471,339.308,358.965,171.253,48.988,159.617
C04483=1022.463,339.061,359.001,171.247,48.989,159.617
C04484=1022.456,338.813,359.037,171.240,48.990,159.616
C04485=1022.449,338.567,359.073,171.233,48.992,159.615
C04486=1022.441,338.319,359.109,171.227,48.993,159.615
C04487=1022.433,338.072,359.146,171.220,48.995,159.614
C04488=1022.427,337.835,359.180,171.214,48.996,159.613
C04489=1022.420,337.599,359.215,171.207,48.997,159.613
C04490=1022.413,337.363,359.248,171.201,48.998,159.612
C04491=1022.406,337.127,359.283,171.196,48.999,159.611
C04492=1022.399,336.891,359.317,171.190,49.001,159.611
C04493=1022.392,336.655,359.351,171.183,49.003,159.610
C04494=1022.385,336.418,359.386,171.177,49.004,159.610
C04495=1022.378,336.181,359.420,171.170,49.005,159.609
C04496=1022.371,335.935,359.456,171.164,49.006,159.608
C04497=1022.363,335.687,359.492,171.158,49.008,159.608
C04498=1022.357,335.440,359.527,171.152,49.010,159.607
C04499=1022.349,335.192,359.563,171.145,49.011,159.607
C04500=1022.342,334.945,359.598,171.138,49.013,159.606
C04501=1022.334,334.698,359.634,171.132,49.014,159.605
C04502=1022.327,334.451,359.670,171.126,49.016,159.605
C04503=1022.320,334.203,359.706,171.119,49.017,159.604
C04504=1022.313,333.956,359.742,171.113,49.018,159.603
C04505=1022.306,333.709,359.777,171.107,49.020,159.603
C04506=1022.299,333.461,359.812,171.100,49.022,159.602
C04507=1022.292,333.214,359.848,171.094,49.023,159.602
C04508=1022.284,332.966,359.884,171.088,49.025,159.601
C04509=1022.277,332.719,359.919,171.082,49.026,159.600
C04510=1022.270,332.472,359.954,171.076,49.028,159.600
C04511=1022.262,332.224,359.990,171.068,49.030,159.599
C04512=1022.256,331.977,360.025,171.062,49.031,159.599
C04513=1022.248,331.730,360.060,171.056,49.033,159.598
C04514=1022.240,331.482,360.095,171.050,49.035,159.598
C04515=1022.234,331.235,360.131,171.044,49.037,159.597
C04516=1022.227,330.987,360.166,171.037,49.038,159.597
C04517=1022.220,330.739,360.201,171.031,49.040,159.596
C04518=1022.212,330.492,360.236,171.025,49.041,159.595
C04519=1022.205,330.245,360.271,171.019,49.043,159.595
C04520=1022.198,329.997,360.307,171.013,49.045,159.594
C04521=1022.191,329.750,360.342,171.006,49.046,159.594
C04522=1022.183,329.503,360.377,171.000,49.048,159.593
C04523=1022.177,329.256,360.412,170.994,49.050,159.593
C04524=1022.169,329.008,360.447,170.988,49.052,159.592
C04525=1022.162,328.760,360.483,170.982,49.053,159.592
C04526=1022.155,328.513,360.517,170.975,49.055,159.591
C04527=1022.148,328.266,360.552,170.969,49.057,159.591
C04528=1022.141,328.018,360.587,170.963,49.059,159.590
C04529=1022.135,327.771,360.622,170.956,49.061,159.590
C04530=1022.127,327.523,360.657,170.950,49.062,159.589
C04531=1022.120,327.275,360.692,170.944,49.064,159.589
C04532=1022.113,327.028,360.727,170.938,49.066,159.588
C04533=1022.106,326.781,360.761,170.932,49.068,159.588
C04534=1022.099,326.534,360.797,170.926,49.070,159.587
C04535=1022.092,326.286,360.830,170.920,49.072,159.587
C04536=1022.084,326.039,360.865,170.914,49.074,159.586
C04537=1022.077,325.790,360.900,170.908,49.076,159.586
C04538=1022.070,325.543,360.934,170.902,49.078,159.585
C04539=1022.062,325.296,360.969,170.896,49.080,159.585
C04540=1022.056,325.048,361.003,170.890,49.082,159.584
C04541=1022.048,324.801,361.038,170.884,49.083,159.584
C04542=1022.041,324.553,361.072,170.878,49.085,159.584
C04543=1022.034,324.306,361.107,170.872,49.087,159.583
C04544=1022.027,324.058,361.141,170.866,49.090,159.583
C04545=1022.020,323.811,361.175,170.860,49.092,159.582
C04546=1022.012,323.564,361.209,170.854,49.094,159.582
C04547=1022.006,323.316,361.243,170.848,49.096,159.581
C04548=1021.999,323.078,361.277,170.842,49.098,159.581
C04549=1021.992,322.839,361.310,170.837,49.100,159.581
C04550=1021.985,322.601,361.343,170.831,49.102,159.580
C04551=1021.978,322.362,361.376,170.825,49.104,159.580
C04552=1021.971,322.124,361.409,170.819,49.106,159.579
C04553=1021.964,321.885,361.442,170.814,49.108,159.579
C04554=1021.958,321.646,361.475,170.808,49.110,159.579
C04555=1021.951,321.408,361.508,170.803,49.112,159.578
C04556=1021.944,321.161,361.541,170.797,49.114,159.578
C04557=1021.937,320.913,361.575,170.791,49.116,159.577
C04558=1021.930,320.666,361.610,170.785,49.118,159.577
C04559=1021.923,320.418,361.644,170.779,49.121,159.577
C04560=1021.916,320.170,361.678,170.773,49.122,159.576
C04561=1021.909,319.922,361.712,170.767,49.124,159.576
C04562=1021.902,319.675,361.746,170.762,49.127,159.575
C04563=1021.895,319.428,361.781,170.756,49.129,159.575
C04564=1021.888,319.181,361.814,170.750,49.131,159.575
C04565=1021.882,318.933,361.849,170.744,49.133,159.574
C04566=1021.874,318.685,361.882,170.738,49.135,159.574
C04567=1021.867,318.437,361.916,170.732,49.138,159.574
C04568=1021.861,318.189,361.951,170.726,49.140,159.573
C04569=1021.854,317.942,361.984,170.720,49.142,159.573
C04570=1021.847,317.695,362.018,170.714,49.144,159.572
C04571=1021.840,317.447,362.052,170.709,49.147,159.572
C04572=1021.833,317.199,362.086,170.703,49.149,159.572
C04573=1021.827,316.952,362.120,170.698,49.151,159.571
C04574=1021.819,316.704,362.154,170.692,49.153,159.571
C04575=1021.812,316.457,362.187,170.686,49.155,159.571
C04576=1021.806,316.209,362.221,170.681,49.158,159.570
C04577=1021.799,315.962,362.255,170.675,49.160,159.570
C04578=1021.792,315.714,362.289,170.669,49.162,159.570
C04579=1021.786,315.466,362.322,170.663,49.165,159.569
C04580=1021.779,315.218,362.356,170.657,49.167,159.569
C04581=1021.772,314.971,362.390,170.651,49.169,159.569
C04582=1021.765,314.724,362.423,170.647,49.172,159.568
C04583=1021.759,314.476,362.458,170.641,49.174,159.568
C04584=1021.752,314.229,362.491,170.635,49.176,159.568
C04585=1021.745,313.981,362.524,170.629,49.179,159.567
C04586=1021.738,313.733,362.558,170.624,49.181,159.567
C04587=1021.732,313.486,362.592,170.618,49.183,159.567
C04588=1021.725,313.238,362.626,170.612,49.186,159.566
C04589=1021.719,312.990,362.659,170.606,49.188,159.566
C04590=1021.712,312.743,362.693,170.602,49.191,159.566
C04591=1021.706,312.495,362.727,170.596,49.193,159.565
C04592=1021.699,312.247,362.760,170.590,49.195,159.565
C04593=1021.692,312.000,362.793,170.584,49.198,159.565
C04594=1021.685,311.752,362.827,170.579,49.200,159.564
C04595=1021.680,311.505,362.861,170.573,49.203,159.564
C04596=1021.672,311.257,362.894,170.568,49.205,159.564
C04597=1021.666,311.009,362.927,170.563,49.208,159.564
C04598=1021.659,310.762,362.961,170.557,49.210,159.563
C04599=1021.653,310.514,362.994,170.551,49.212,159.563
C04600=1021.647,310.267,363.028,170.545,49.215,159.563
C04601=1021.640,310.018,363.061,170.539,49.217,159.562
C04602=1021.633,309.772,363.094,170.535,49.220,159.562
C04603=1021.626,309.524,363.127,170.529,49.223,159.562
C04604=1021.619,309.276,363.160,170.524,49.225,159.562
C04605=1021.612,309.028,363.192,170.518,49.228,159.562
C04606=1021.605,308.781,363.225,170.512,49.230,159.561
C04607=1021.597,308.533,363.258,170.507,49.233,159.561
C04608=1021.592,308.297,363.289,170.501,49.236,159.561
C04609=1021.585,308.061,363.320,170.497,49.238,159.561
C04610=1021.579,307.826,363.352,170.491,49.241,159.560
C04611=1021.572,307.589,363.383,170.485,49.243,159.560
C04612=1021.565,307.353,363.413,170.481,49.246,159.560
C04613=1021.559,307.117,363.445,170.475,49.249,159.560
C04614=1021.553,306.882,363.476,170.471,49.251,159.560
C04615=1021.546,306.646,363.507,170.465,49.254,159.559
C04616=1021.539,306.398,363.540,170.460,49.257,159.559
C04617=1021.532,306.151,363.572,170.454,49.259,159.559
C04618=1021.526,305.903,363.605,170.448,49.262,159.559
C04619=1021.518,305.655,363.638,170.444,49.265,159.559
C04620=1021.512,305.407,363.670,170.438,49.267,159.558
C04621=1021.506,305.160,363.703,170.433,49.271,159.558
C04622=1021.498,304.912,363.736,170.427,49.273,159.558
C04623=1021.492,304.664,363.768,170.422,49.276,159.558
C04624=1021.486,304.417,363.801,170.416,49.279,159.558
C04625=1021.478,304.168,363.833,170.411,49.282,159.557
C04626=1021.472,303.920,363.866,170.406,49.284,159.557
C04627=1021.465,303.673,363.898,170.401,49.287,159.557
C04628=1021.459,303.426,363.931,170.395,49.290,159.557
C04629=1021.452,303.177,363.964,170.390,49.293,159.557
C04630=1021.445,302.930,363.996,170.384,49.296,159.557
C04631=1021.439,302.682,364.028,170.379,49.299,159.556
C04632=1021.432,302.434,364.060,170.373,49.302,159.556
C04633=1021.425,302.187,364.093,170.369,49.305,159.556
C04634=1021.418,301.939,364.126,170.363,49.307,159.556
C04635=1021.412,301.691,364.157,170.358,49.310,159.556
C04636=1021.405,301.443,364.190,170.352,49.313,159.556
C04637=1021.398,301.196,364.222,170.347,49.316,159.555
C04638=1021.392,300.948,364.254,170.343,49.319,159.555
C04639=1021.386,300.700,364.287,170.337,49.322,159.555
C04640=1021.379,300.453,364.319,170.332,49.325,159.555
C04641=1021.373,300.204,364.351,170.326,49.328,159.555
C04642=1021.365,299.957,364.384,170.321,49.331,159.555
C04643=1021.359,299.709,364.416,170.315,49.334,159.555
C04644=1021.353,299.461,364.448,170.311,49.336,159.554
C04645=1021.346,299.213,364.480,170.305,49.339,159.554
C04646=1021.340,298.965,364.513,170.300,49.343,159.554
C04647=1021.333,298.718,364.545,170.295,49.346,159.554
C04648=1021.327,298.470,364.577,170.290,49.348,159.554
C04649=1021.321,298.222,364.609,170.285,49.351,159.554
C04650=1021.314,297.974,364.641,170.279,49.355,159.554
C04651=1021.308,297.727,364.674,170.274,49.358,159.554
C04652=1021.301,297.479,364.705,170.268,49.360,159.553
C04653=1021.295,297.231,364.738,170.264,49.363,159.553
C04654=1021.288,296.983,364.769,170.259,49.366,159.553
C04655=1021.282,296.735,364.801,170.254,49.370,159.553
C04656=1021.276,296.487,364.834,170.248,49.373,159.553
C04657=1021.269,296.240,364.865,170.244,49.376,159.553
C04658=1021.263,295.992,364.898,170.238,49.378,159.553
C04659=1021.256,295.744,364.930,170.233,49.382,159.553
C04660=1021.250,295.496,364.962,170.228,49.385,159.553
C04661=1021.244,295.248,364.994,170.223,49.388,159.553
C04662=1021.237,295.000,365.026,170.218,49.391,159.552
C04663=1021.231,294.752,365.058,170.213,49.394,159.552
C04664=1021.224,294.504,365.089,170.207,49.397,159.552
C04665=1021.218,294.257,365.122,170.203,49.400,159.552
C04666=1021.212,294.009,365.153,170.198,49.404,159.552
C04667=1021.206,293.761,365.185,170.192,49.407,159.552
C04668=1021.200,293.534,365.214,170.188,49.410,159.552
C04669=1021.195,293.306,365.244,170.182,49.412,159.552
C04670=1021.188,293.079,365.272,170.178,49.415,159.552
C04671=1021.182,292.852,365.302,170.174,49.418,159.552
C04672=1021.176,292.625,365.330,170.169,49.421,159.552
C04673=1021.171,292.398,365.359,170.164,49.424,159.552
C04674=1021.164,292.171,365.388,170.160,49.427,159.552
C04675=1021.159,291.944,365.417,170.155,49.430,159.552
C04676=1021.152,291.696,365.449,170.150,49.433,159.551
C04677=1021.145,291.448,365.480,170.145,49.437,159.552
C04678=1021.139,291.201,365.511,170.140,49.440,159.551
C04679=1021.132,290.953,365.542,170.135,49.444,159.551
C04680=1021.126,290.705,365.574,170.130,49.447,159.551
C04681=1021.119,290.457,365.605,170.125,49.450,159.551
C04682=1021.113,290.209,365.637,170.120,49.454,159.551
C04683=1021.107,289.960,365.668,170.115,49.457,159.551
C04684=1021.100,289.713,365.699,170.110,49.461,159.551
C04685=1021.094,289.465,365.731,170.105,49.464,159.551
C04686=1021.087,289.217,365.762,170.100,49.467,159.551
C04687=1021.080,288.969,365.793,170.095,49.471,159.551
C04688=1021.074,288.721,365.824,170.090,49.474,159.551
C04689=1021.068,288.474,365.855,170.084,49.477,159.551
C04690=1021.061,288.226,365.887,170.080,49.481,159.551
C04691=1021.055,287.977,365.917,170.075,49.484,159.551
C04692=1021.049,287.729,365.949,170.070,49.488,159.551
C04693=1021.043,287.482,365.980,170.065,49.491,159.551
C04694=1021.036,287.233,366.011,170.061,49.495,159.551
C04695=1021.029,286.985,366.043,170.056,49.498,159.551
C04696=1021.023,286.738,366.074,170.051,49.502,159.551
C04697=1021.017,286.490,366.104,170.045,49.505,159.551
C04698=1021.010,286.242,366.136,170.040,49.509,159.551
C04699=1021.004,285.994,366.166,170.036,49.512,159.551
C04700=1020.998,285.746,366.198,170.031,49.516,159.551
C04701=1020.991,285.497,366.228,170.026,49.519,159.551
C04702=1020.984,285.250,366.260,170.021,49.523,159.551
C04703=1020.979,285.002,366.290,170.017,49.526,159.551
C04704=1020.971,284.754,366.321,170.012,49.530,159.551
C04705=1020.965,284.506,366.352,170.007,49.534,159.552
C04706=1020.959,284.258,366.382,170.001,49.537,159.551
C04707=1020.952,284.010,366.413,169.996,49.541,159.552
C04708=1020.946,283.761,366.444,169.991,49.545,159.552
C04709=1020.939,283.514,366.474,169.987,49.548,159.552
C04710=1020.932,283.266,366.505,169.982,49.551,159.552
C04711=1020.927,283.018,366.536,169.977,49.555,159.552
C04712=1020.920,282.770,366.566,169.972,49.559,159.552
C04713=1020.914,282.522,366.598,169.967,49.563,159.552
C04714=1020.907,282.274,366.628,169.963,49.566,159.552
C04715=1020.901,282.026,366.658,169.958,49.570,159.552
C04716=1020.895,281.778,366.689,169.953,49.574,159.552
C04717=1020.888,281.529,366.719,169.948,49.578,159.552
C04718=1020.882,281.281,366.751,169.943,49.582,159.552
C04719=1020.875,281.034,366.781,169.939,49.585,159.552
C04720=1020.869,280.785,366.811,169.934,49.589,159.552
C04721=1020.863,280.538,366.842,169.929,49.592,159.553
C04722=1020.856,280.289,366.872,169.924,49.596,159.553
C04723=1020.851,280.041,366.903,169.920,49.600,159.553
C04724=1020.843,279.794,366.934,169.915,49.604,159.553
C04725=1020.837,279.546,366.964,169.910,49.608,159.553
C04726=1020.831,279.297,366.995,169.905,49.611,159.553
C04727=1020.825,279.049,367.025,169.900,49.615,159.553
C04728=1020.819,278.828,367.051,169.896,49.618,159.553
C04729=1020.814,278.608,367.079,169.892,49.622,159.553
C04730=1020.808,278.386,367.106,169.888,49.625,159.553
C04731=1020.803,278.166,367.133,169.884,49.629,159.553
C04732=1020.797,277.944,367.160,169.880,49.632,159.554
C04733=1020.791,277.723,367.187,169.876,49.635,159.554
C04734=1020.786,277.503,367.214,169.871,49.639,159.554
C04735=1020.780,277.281,367.241,169.867,49.643,159.554
C04736=1020.774,277.033,367.272,169.863,49.646,159.554
C04737=1020.767,276.785,367.302,169.858,49.650,159.554
C04738=1020.761,276.537,367.332,169.853,49.654,159.554
C04739=1020.755,276.290,367.362,169.848,49.658,159.554
C04740=1020.748,276.041,367.393,169.843,49.662,159.554
C04741=1020.742,275.793,367.422,169.839,49.665,159.555
C04742=1020.736,275.544,367.453,169.834,49.669,159.555
C04743=1020.730,275.297,367.483,169.829,49.673,159.555
C04744=1020.723,275.049,367.513,169.824,49.678,159.555
C04745=1020.717,274.801,367.543,169.820,49.682,159.555
C04746=1020.711,274.552,367.572,169.816,49.685,159.555
C04747=1020.705,274.305,367.603,169.811,49.689,159.555
C04748=1020.698,274.056,367.633,169.806,49.693,159.555
C04749=1020.692,273.808,367.663,169.801,49.698,159.556
C04750=1020.686,273.560,367.692,169.796,49.702,159.556
C04751=1020.679,273.312,367.723,169.792,49.705,159.556
C04752=1020.673,273.064,367.752,169.788,49.710,159.556
C04753=1020.667,272.816,367.782,169.783,49.714,159.556
C04754=1020.660,272.568,367.812,169.778,49.718,159.556
C04755=1020.654,272.319,367.842,169.773,49.722,159.557
C04756=1020.648,272.072,367.872,169.769,49.726,159.557
C04757=1020.642,271.823,367.902,169.764,49.730,159.557
C04758=1020.635,271.575,367.932,169.760,49.734,159.557
C04759=1020.629,271.327,367.961,169.755,49.738,159.557
C04760=1020.623,271.079,367.991,169.750,49.742,159.557
C04761=1020.616,270.830,368.020,169.746,49.746,159.558
C04762=1020.611,270.583,368.051,169.741,49.750,159.558
C04763=1020.604,270.334,368.080,169.737,49.755,159.558
C04764=1020.598,270.086,368.111,169.732,49.759,159.558
C04765=1020.592,269.838,368.140,169.727,49.763,159.558
C04766=1020.585,269.590,368.169,169.723,49.767,159.559
C04767=1020.580,269.342,368.199,169.718,49.771,159.559
C04768=1020.573,269.094,368.228,169.714,49.776,159.559
C04769=1020.566,268.845,368.258,169.709,49.779,159.559
C04770=1020.561,268.597,368.288,169.704,49.784,159.559
C04771=1020.554,268.349,368.317,169.701,49.788,159.560
C04772=1020.548,268.101,368.347,169.696,49.792,159.560
C04773=1020.541,267.853,368.376,169.691,49.797,159.560
C04774=1020.535,267.604,368.406,169.686,49.801,159.560
C04775=1020.529,267.357,368.435,169.682,49.805,159.561
C04776=1020.523,267.108,368.464,169.677,49.810,159.561
C04777=1020.516,266.860,368.493,169.673,49.814,159.561
C04778=1020.511,266.612,368.523,169.669,49.818,159.561
C04779=1020.504,266.363,368.552,169.664,49.822,159.561
C04780=1020.498,266.116,368.582,169.659,49.827,159.562
C04781=1020.491,265.867,368.611,169.654,49.831,159.562
C04782=1020.486,265.619,368.641,169.651,49.835,159.562
C04783=1020.479,265.371,368.670,169.646,49.839,159.562
C04784=1020.473,265.123,368.699,169.641,49.844,159.563
C04785=1020.467,264.875,368.728,169.637,49.849,159.563
C04786=1020.461,264.626,368.757,169.632,49.853,159.563
C04787=1020.454,264.378,368.786,169.627,49.857,159.563
C04788=1020.449,264.159,368.813,169.624,49.861,159.564
C04789=1020.444,263.941,368.838,169.620,49.865,159.564
C04790=1020.437,263.722,368.864,169.616,49.869,159.564
C04791=1020.432,263.504,368.889,169.612,49.873,159.564
C04792=1020.427,263.285,368.916,169.608,49.877,159.565
C04793=1020.421,263.065,368.941,169.604,49.881,159.565
C04794=1020.416,262.847,368.966,169.600,49.885,159.565
C04795=1020.410,262.629,368.992,169.596,49.888,159.565
C04796=1020.404,262.381,369.021,169.591,49.893,159.565
C04797=1020.399,262.132,369.050,169.588,49.897,159.566
C04798=1020.392,261.884,369.080,169.583,49.902,159.566
C04799=1020.385,261.635,369.109,169.579,49.906,159.566
C04800=1020.379,261.387,369.138,169.574,49.911,159.567
C04801=1020.373,261.139,369.166,169.570,49.916,159.567
C04802=1020.367,260.890,369.195,169.565,49.920,159.567
C04803=1020.361,260.642,369.224,169.561,49.925,159.568
C04804=1020.354,260.394,369.253,169.557,49.929,159.568
C04805=1020.348,260.146,369.282,169.552,49.934,159.568
C04806=1020.342,259.898,369.311,169.548,49.938,159.568
C04807=1020.337,259.650,369.339,169.543,49.943,159.569
C04808=1020.330,259.402,369.368,169.539,49.948,159.569
C04809=1020.323,259.153,369.397,169.534,49.952,159.569
C04810=1020.317,258.904,369.426,169.530,49.957,159.569
C04811=1020.310,258.657,369.454,169.525,49.962,159.570
C04812=1020.304,258.408,369.482,169.521,49.967,159.570
C04813=1020.298,258.160,369.511,169.517,49.971,159.571
C04814=1020.292,257.912,369.539,169.513,49.976,159.571
C04815=1020.285,257.664,369.568,169.508,49.980,159.571
C04816=1020.279,257.415,369.596,169.504,49.986,159.572
C04817=1020.272,257.167,369.625,169.499,49.990,159.572
C04818=1020.266,256.919,369.653,169.495,49.995,159.572
C04819=1020.260,256.670,369.682,169.491,50.000,159.573
C04820=1020.254,256.422,369.710,169.486,50.005,159.573
C04821=1020.247,256.174,369.739,169.482,50.009,159.573
C04822=1020.241,255.925,369.767,169.477,50.014,159.573
C04823=1020.234,255.677,369.795,169.473,50.019,159.574
C04824=1020.228,255.428,369.824,169.468,50.024,159.574
C04825=1020.222,255.180,369.853,169.465,50.028,159.575
C04826=1020.216,254.932,369.881,169.460,50.033,159.575
C04827=1020.209,254.684,369.910,169.456,50.038,159.575
C04828=1020.204,254.436,369.938,169.451,50.043,159.576
C04829=1020.197,254.187,369.965,169.447,50.048,159.576
C04830=1020.191,253.939,369.994,169.443,50.053,159.576
C04831=1020.185,253.690,370.023,169.438,50.058,159.577
C04832=1020.178,253.442,370.050,169.434,50.062,159.577
C04833=1020.172,253.194,370.079,169.429,50.067,159.577
C04834=1020.166,252.945,370.108,169.425,50.072,159.578
C04835=1020.160,252.697,370.135,169.421,50.077,159.578
C04836=1020.154,252.449,370.164,169.417,50.082,159.579
C04837=1020.148,252.200,370.192,169.413,50.087,159.579
C04838=1020.141,251.952,370.220,169.409,50.092,159.579
C04839=1020.135,251.703,370.249,169.404,50.097,159.580
C04840=1020.130,251.456,370.277,169.400,50.102,159.580
C04841=1020.123,251.207,370.305,169.395,50.106,159.580
C04842=1020.117,250.959,370.333,169.391,50.112,159.581
C04843=1020.111,250.710,370.362,169.387,50.116,159.581
C04844=1020.105,250.463,370.390,169.383,50.122,159.582
C04845=1020.099,250.214,370.418,169.378,50.126,159.582
C04846=1020.093,249.965,370.446,169.374,50.132,159.582
C04847=1020.086,249.717,370.474,169.370,50.136,159.583
C04848=1020.082,249.498,370.499,169.366,50.141,159.583
C04849=1020.076,249.278,370.525,169.362,50.145,159.583
C04850=1020.071,249.059,370.549,169.359,50.149,159.584
C04851=1020.065,248.839,370.574,169.355,50.154,159.584
C04852=1020.059,248.619,370.599,169.351,50.159,159.585
C04853=1020.054,248.400,370.623,169.347,50.163,159.585
C04854=1020.049,248.180,370.648,169.344,50.167,159.585
C04855=1020.043,247.961,370.673,169.340,50.172,159.586
C04856=1020.037,247.713,370.701,169.336,50.176,159.586
C04857=1020.031,247.464,370.730,169.332,50.182,159.586
C04858=1020.025,247.216,370.757,169.327,50.187,159.587
C04859=1020.019,246.967,370.785,169.323,50.192,159.587
C04860=1020.013,246.719,370.814,169.319,50.197,159.588
C04861=1020.007,246.471,370.841,169.315,50.202,159.588
C04862=1020.001,246.222,370.869,169.310,50.207,159.588
C04863=1019.996,245.974,370.897,169.307,50.212,159.589
C04864=1019.989,245.726,370.925,169.303,50.217,159.589
C04865=1019.983,245.477,370.953,169.298,50.222,159.590
C04866=1019.978,245.229,370.981,169.294,50.227,159.590
C04867=1019.971,244.980,371.009,169.290,50.233,159.591
C04868=1019.966,244.732,371.037,169.286,50.238,159.591
C04869=1019.959,244.484,371.065,169.281,50.243,159.591
C04870=1019.954,244.235,371.093,169.277,50.248,159.592
C04871=1019.948,243.987,371.121,169.273,50.253,159.592
C04872=1019.941,243.739,371.149,169.269,50.259,159.593
C04873=1019.936,243.490,371.176,169.266,50.264,159.593
C04874=1019.931,243.241,371.204,169.261,50.268,159.593
C04875=1019.924,242.994,371.232,169.257,50.273,159.594
C04876=1019.918,242.745,371.259,169.253,50.279,159.594
C04877=1019.912,242.496,371.288,169.248,50.284,159.595
C04878=1019.906,242.248,371.314,169.244,50.289,159.595
C04879=1019.899,242.000,371.342,169.240,50.295,159.596
C04880=1019.894,241.751,371.370,169.236,50.300,159.596
C04881=1019.888,241.502,371.397,169.232,50.305,159.597
C04882=1019.882,241.255,371.424,169.228,50.311,159.597
C04883=1019.876,241.006,371.453,169.224,50.316,159.598
C04884=1019.870,240.758,371.479,169.219,50.321,159.598
C04885=1019.863,240.509,371.507,169.215,50.327,159.599
C04886=1019.858,240.261,371.535,169.211,50.332,159.599
C04887=1019.851,240.012,371.562,169.207,50.337,159.600
C04888=1019.846,239.764,371.590,169.203,50.343,159.600
C04889=1019.839,239.516,371.618,169.199,50.348,159.600
C04890=1019.834,239.267,371.644,169.194,50.353,159.601
C04891=1019.827,239.019,371.672,169.191,50.359,159.602
C04892=1019.822,238.770,371.699,169.187,50.365,159.602
C04893=1019.815,238.522,371.727,169.182,50.370,159.603
C04894=1019.809,238.273,371.754,169.178,50.376,159.603
C04895=1019.803,238.025,371.782,169.174,50.381,159.603
C04896=1019.797,237.776,371.808,169.170,50.387,159.604
C04897=1019.791,237.527,371.835,169.166,50.392,159.605
C04898=1019.785,237.280,371.863,169.162,50.398,159.605
C04899=1019.778,237.031,371.890,169.158,50.403,159.606
C04900=1019.772,236.783,371.917,169.154,50.409,159.606
C04901=1019.766,236.534,371.944,169.150,50.414,159.607
C04902=1019.760,236.285,371.971,169.146,50.420,159.607
C04903=1019.755,236.037,371.999,169.142,50.426,159.608
C04904=1019.748,235.788,372.026,169.138,50.431,159.608
C04905=1019.742,235.540,372.052,169.133,50.437,159.609
C04906=1019.736,235.292,372.080,169.129,50.443,159.609
C04907=1019.730,235.043,372.107,169.125,50.448,159.610
C04908=1019.724,234.820,372.130,169.122,50.453,159.610
C04909=1019.719,234.598,372.154,169.118,50.458,159.611
C04910=1019.713,234.375,372.179,169.115,50.463,159.611
C04911=1019.707,234.152,372.203,169.111,50.468,159.612
C04912=1019.703,233.930,372.227,169.107,50.473,159.612
C04913=1019.697,233.707,372.251,169.104,50.478,159.613
C04914=1019.691,233.484,372.275,169.100,50.484,159.613
C04915=1019.686,233.261,372.299,169.096,50.489,159.614
C04916=1019.680,233.013,372.327,169.092,50.494,159.614
C04917=1019.674,232.764,372.354,169.089,50.500,159.615
C04918=1019.668,232.516,372.380,169.084,50.505,159.615
C04919=1019.662,232.267,372.407,169.081,50.511,159.616
C04920=1019.656,232.019,372.434,169.076,50.517,159.616
C04921=1019.650,231.770,372.461,169.072,50.523,159.617
C04922=1019.644,231.522,372.488,169.068,50.528,159.617
C04923=1019.638,231.273,372.515,169.064,50.534,159.618
C04924=1019.632,231.025,372.542,169.060,50.540,159.619
C04925=1019.626,230.776,372.569,169.056,50.546,159.619
C04926=1019.620,230.528,372.595,169.052,50.551,159.620
C04927=1019.614,230.279,372.622,169.048,50.557,159.620
C04928=1019.608,230.031,372.649,169.044,50.563,159.621
C04929=1019.602,229.782,372.676,169.040,50.569,159.622
C04930=1019.596,229.534,372.702,169.037,50.575,159.622
C04931=1019.590,229.285,372.729,169.033,50.581,159.623
C04932=1019.585,229.037,372.755,169.028,50.586,159.623
C04933=1019.578,228.788,372.782,169.024,50.593,159.624
C04934=1019.572,228.540,372.809,169.020,50.599,159.625
C04935=1019.566,228.291,372.835,169.016,50.604,159.625
C04936=1019.560,228.043,372.862,169.012,50.610,159.626
C04937=1019.554,227.794,372.889,169.009,50.616,159.626
C04938=1019.548,227.546,372.916,169.004,50.621,159.627
C04939=1019.542,227.297,372.942,169.001,50.627,159.627
C04940=1019.536,227.049,372.968,168.997,50.634,159.628
C04941=1019.529,226.800,372.995,168.992,50.640,159.629
C04942=1019.524,226.551,373.021,168.988,50.645,159.629
C04943=1019.518,226.303,373.048,168.984,50.651,159.630
C04944=1019.512,226.055,373.074,168.981,50.657,159.630
C04945=1019.506,225.806,373.101,168.977,50.663,159.631
C04946=1019.499,225.557,373.126,168.972,50.670,159.632
C04947=1019.493,225.309,373.153,168.969,50.676,159.632
C04948=1019.488,225.060,373.180,168.965,50.682,159.633
C04949=1019.481,224.812,373.206,168.961,50.688,159.634
C04950=1019.476,224.563,373.232,168.957,50.694,159.634
C04951=1019.468,224.314,373.258,168.954,50.700,159.635
C04952=1019.463,224.066,373.285,168.949,50.707,159.636
C04953=1019.457,223.817,373.311,168.945,50.713,159.636
C04954=1019.451,223.569,373.337,168.941,50.719,159.637
C04955=1019.445,223.321,373.363,168.938,50.725,159.638
C04956=1019.439,223.072,373.389,168.934,50.731,159.638
C04957=1019.432,222.823,373.416,168.929,50.737,159.639
C04958=1019.427,222.574,373.441,168.926,50.743,159.640
C04959=1019.420,222.326,373.468,168.922,50.749,159.640
C04960=1019.415,222.078,373.494,168.918,50.755,159.641
C04961=1019.408,221.829,373.520,168.913,50.762,159.641
C04962=1019.403,221.581,373.546,168.910,50.768,159.642
C04963=1019.397,221.332,373.572,168.906,50.774,159.643
C04964=1019.391,221.084,373.598,168.902,50.780,159.643
C04965=1019.385,220.835,373.624,168.899,50.786,159.644
C04966=1019.378,220.586,373.651,168.894,50.793,159.645
C04967=1019.372,220.337,373.677,168.890,50.799,159.645
C04968=1019.367,220.111,373.701,168.887,50.804,159.646
C04969=1019.362,219.884,373.724,168.883,50.810,159.646
C04970=1019.356,219.657,373.748,168.880,50.816,159.647
C04971=1019.351,219.430,373.772,168.877,50.822,159.648
C04972=1019.346,219.203,373.796,168.873,50.827,159.648
C04973=1019.340,218.977,373.819,168.869,50.833,159.649
C04974=1019.334,218.749,373.843,168.865,50.839,159.650
C04975=1019.329,218.523,373.867,168.862,50.844,159.650
C04976=1019.324,218.274,373.893,168.859,50.850,159.651
C04977=1019.317,218.026,373.919,168.854,50.858,159.652
C04978=1019.311,217.777,373.944,168.851,50.864,159.652
C04979=1019.305,217.529,373.970,168.847,50.870,159.653
C04980=1019.299,217.280,373.996,168.842,50.877,159.654
C04981=1019.293,217.031,374.021,168.839,50.883,159.654
C04982=1019.286,216.783,374.047,168.835,50.889,159.655
C04983=1019.281,216.534,374.073,168.831,50.896,159.656
C04984=1019.275,216.285,374.099,168.827,50.902,159.657
C04985=1019.269,216.037,374.124,168.824,50.909,159.657
C04986=1019.262,215.789,374.150,168.820,50.915,159.658
C04987=1019.257,215.540,374.176,168.815,50.921,159.659
C04988=1019.250,215.291,374.201,168.812,50.928,159.659
C04989=1019.244,215.042,374.227,168.808,50.934,159.660
C04990=1019.239,214.793,374.253,168.804,50.941,159.661
C04991=1019.232,214.545,374.279,168.800,50.948,159.662
C04992=1019.226,214.297,374.304,168.797,50.954,159.662
C04993=1019.220,214.048,374.330,168.792,50.961,159.663
C04994=1019.214,213.799,374.355,168.789,50.968,159.664
C04995=1019.208,213.550,374.381,168.785,50.974,159.665
C04996=1019.202,213.302,374.406,168.781,50.981,159.665
C04997=1019.196,213.053,374.433,168.777,50.987,159.666
C04998=1019.190,212.805,374.458,168.774,50.994,159.667
C04999=1019.184,212.556,374.483,168.769,51.000,159.667
C05000=1019.179,212.308,374.509,168.766,51.007,159.668
C05001=1019.173,212.059,374.534,168.762,51.013,159.669
C05002=1019.166,211.810,374.560,168.758,51.020,159.670
C05003=1019.160,211.562,374.585,168.754,51.026,159.670
C05004=1019.155,211.313,374.611,168.751,51.033,159.671
C05005=1019.149,211.064,374.636,168.747,51.040,159.672
C05006=1019.142,210.815,374.661,168.743,51.046,159.673
C05007=1019.137,210.566,374.687,168.740,51.053,159.674
C05008=1019.131,210.318,374.713,168.735,51.060,159.674
C05009=1019.125,210.070,374.738,168.732,51.066,159.675
C05010=1019.119,209.821,374.763,168.728,51.074,159.676
C05011=1019.113,209.572,374.788,168.724,51.080,159.676
C05012=1019.107,209.324,374.814,168.721,51.087,159.677
C05013=1019.101,209.075,374.840,168.716,51.094,159.678
C05014=1019.095,208.826,374.865,168.713,51.100,159.679
C05015=1019.089,208.578,374.890,168.708,51.107,159.679
C05016=1019.083,208.330,374.915,168.705,51.114,159.680
C05017=1019.077,208.081,374.941,168.702,51.121,159.681
C05018=1019.071,207.832,374.966,168.698,51.128,159.682
C05019=1019.065,207.583,374.991,168.694,51.135,159.683
C05020=1019.058,207.334,375.016,168.690,51.141,159.683
C05021=1019.053,207.086,375.041,168.686,51.148,159.684
C05022=1019.047,206.838,375.066,168.682,51.155,159.685
C05023=1019.040,206.589,375.092,168.679,51.162,159.686
C05024=1019.035,206.340,375.116,168.676,51.169,159.687
C05025=1019.029,206.092,375.141,168.671,51.176,159.688
C05026=1019.023,205.843,375.167,168.668,51.183,159.688
C05027=1019.016,205.594,375.192,168.664,51.190,159.689
C05028=1019.011,205.369,375.214,168.660,51.196,159.690
C05029=1019.006,205.143,375.238,168.658,51.202,159.691
C05030=1019.000,204.918,375.260,168.654,51.208,159.691
C05031=1018.995,204.692,375.282,168.651,51.215,159.692
C05032=1018.989,204.467,375.305,168.647,51.221,159.693
C05033=1018.984,204.241,375.327,168.644,51.228,159.694
C05034=1018.978,204.017,375.350,168.640,51.234,159.694
C05035=1018.973,203.791,375.373,168.637,51.241,159.695
C05036=1018.951,202.702,375.475,168.172,51.145,159.591
C05037=1018.947,202.484,375.495,168.169,51.152,159.592
C05038=1018.941,202.266,375.516,168.164,51.159,159.593
C05039=1018.937,202.048,375.537,168.160,51.166,159.593
C05040=1018.932,201.799,375.560,168.156,51.174,159.594
C05041=1018.927,201.551,375.583,168.151,51.182,159.595
C05042=1018.922,201.302,375.606,168.147,51.190,159.596
C05043=1018.917,201.052,375.630,168.142,51.198,159.597
C05044=1018.912,200.804,375.652,168.138,51.206,159.598
C05045=1018.907,200.555,375.676,168.133,51.214,159.598
C05046=1018.902,200.306,375.700,168.129,51.221,159.599
C05047=1018.897,200.057,375.723,168.124,51.230,159.600
C05048=1018.892,199.808,375.746,168.120,51.238,159.601
C05049=1018.887,199.559,375.769,168.116,51.245,159.602
C05050=1018.882,199.311,375.792,168.111,51.254,159.603
C05051=1018.877,199.062,375.815,168.106,51.262,159.604
C05052=1018.870,198.742,375.844,168.101,51.272,159.605
C05053=1018.864,198.423,375.874,168.096,51.283,159.606
C05054=1018.857,198.104,375.903,168.089,51.293,159.607
C05055=1018.850,197.784,375.932,168.084,51.303,159.608
C05056=1018.845,197.535,375.955,168.080,51.312,159.609
C05057=1018.840,197.287,375.978,168.076,51.320,159.610
C05058=1018.834,197.037,376.000,168.071,51.328,159.611
C05059=1018.829,196.788,376.023,168.067,51.336,159.612
C05060=1018.824,196.540,376.046,168.062,51.344,159.613
C05061=1018.818,196.291,376.069,168.058,51.352,159.614
C05062=1018.813,196.042,376.092,168.053,51.361,159.614
C05063=1018.809,195.793,376.115,168.049,51.368,159.615
C05064=1018.803,195.544,376.138,168.044,51.377,159.616
C05065=1018.798,195.295,376.160,168.041,51.385,159.617
C05066=1018.793,195.046,376.183,168.036,51.393,159.618
C05067=1018.788,194.798,376.206,168.032,51.402,159.619
C05068=1018.783,194.548,376.228,168.027,51.410,159.620
C05069=1018.778,194.300,376.251,168.023,51.418,159.621
C05070=1018.773,194.050,376.273,168.018,51.426,159.621
C05071=1018.767,193.801,376.296,168.015,51.434,159.622
C05072=1018.763,193.553,376.319,168.010,51.442,159.623
C05073=1018.757,193.303,376.342,168.006,51.450,159.624
C05074=1018.752,193.055,376.364,168.001,51.458,159.625
C05075=1018.747,192.805,376.387,167.997,51.466,159.626
C05076=1018.742,192.557,376.410,167.993,51.474,159.627
C05077=1018.737,192.308,376.432,167.989,51.483,159.628
C05078=1018.732,192.059,376.455,167.985,51.491,159.629
C05079=1018.727,191.810,376.477,167.980,51.499,159.629
C05080=1018.722,191.562,376.500,167.976,51.507,159.630
C05081=1018.717,191.313,376.522,167.971,51.516,159.631
C05082=1018.712,191.064,376.545,167.967,51.524,159.632
C05083=1018.707,190.815,376.567,167.963,51.532,159.633
C05084=1018.702,190.566,376.590,167.958,51.540,159.634
C05085=1018.697,190.317,376.612,167.955,51.548,159.635
C05086=1018.692,190.068,376.635,167.950,51.557,159.636
C05087=1018.687,189.819,376.657,167.946,51.565,159.637
C05088=1018.683,189.570,376.680,167.942,51.573,159.638
C05089=1018.677,189.321,376.703,167.938,51.581,159.638
C05090=1018.672,189.072,376.725,167.934,51.589,159.639
C05091=1018.666,188.823,376.748,167.930,51.597,159.640
C05092=1018.662,188.574,376.770,167.925,51.605,159.641
C05093=1018.658,188.325,376.792,167.921,51.613,159.642
C05094=1018.652,188.076,376.815,167.918,51.622,159.643
C05095=1018.648,187.827,376.837,167.913,51.630,159.644
C05096=1018.641,187.547,376.863,167.908,51.639,159.645
C05097=1018.637,187.266,376.888,167.904,51.648,159.646
C05098=1018.630,186.985,376.913,167.898,51.657,159.647
C05099=1018.625,186.704,376.938,167.894,51.666,159.648
C05100=1018.620,186.456,376.960,167.890,51.674,159.649
C05101=1018.615,186.206,376.983,167.887,51.683,159.650
C05102=1018.611,185.957,377.005,167.882,51.691,159.651
C05103=1018.606,185.709,377.028,167.878,51.699,159.652
C05104=1018.601,185.459,377.051,167.874,51.707,159.653
C05105=1018.596,185.210,377.072,167.869,51.716,159.653
C05106=1018.591,184.961,377.094,167.865,51.724,159.654
C05107=1018.585,184.712,377.117,167.862,51.732,159.655
C05108=1018.581,184.463,377.140,167.858,51.740,159.656
C05109=1018.577,184.214,377.162,167.853,51.749,159.657
C05110=1018.572,183.966,377.183,167.849,51.757,159.658
C05111=1018.567,183.716,377.206,167.846,51.765,159.659
C05112=1018.562,183.468,377.229,167.842,51.773,159.660
C05113=1018.557,183.219,377.251,167.837,51.781,159.661
C05114=1018.552,182.970,377.273,167.833,51.789,159.662
C05115=1018.548,182.720,377.295,167.829,51.797,159.663
C05116=1018.543,182.471,377.317,167.826,51.806,159.664
C05117=1018.538,182.223,377.339,167.821,51.814,159.664
C05118=1018.533,181.973,377.362,167.817,51.822,159.665
C05119=1018.528,181.724,377.383,167.813,51.830,159.666
C05120=1018.523,181.475,377.405,167.809,51.839,159.667
C05121=1018.518,181.227,377.427,167.805,51.847,159.668
C05122=1018.512,180.977,377.449,167.802,51.856,159.669
C05123=1018.507,180.729,377.470,167.797,51.864,159.670
C05124=1018.503,180.479,377.492,167.793,51.872,159.671
C05125=1018.497,180.231,377.513,167.789,51.881,159.672
C05126=1018.492,179.981,377.535,167.785,51.889,159.673
C05127=1018.487,179.732,377.557,167.782,51.898,159.674
C05128=1018.481,179.483,377.578,167.777,51.906,159.675
C05129=1018.477,179.234,377.599,167.773,51.915,159.676
C05130=1018.471,178.985,377.622,167.769,51.923,159.677
C05131=1018.466,178.736,377.643,167.765,51.932,159.678
C05132=1018.461,178.487,377.664,167.761,51.940,159.679
C05133=1018.456,178.238,377.685,167.758,51.949,159.680
C05134=1018.451,177.990,377.707,167.753,51.957,159.681
C05135=1018.446,177.739,377.729,167.750,51.966,159.682
C05136=1018.440,177.491,377.750,167.745,51.974,159.683
C05137=1018.435,177.242,377.772,167.741,51.982,159.684
C05138=1018.430,176.993,377.794,167.738,51.991,159.685
C05139=1018.425,176.744,377.814,167.733,51.999,159.686
C05140=1018.420,176.495,377.836,167.730,52.008,159.687
C05141=1018.415,176.245,377.858,167.726,52.016,159.688
C05142=1018.410,175.997,377.879,167.722,52.025,159.689
C05143=1018.405,175.748,377.901,167.718,52.033,159.690
C05144=1018.400,175.499,377.921,167.714,52.042,159.691
C05145=1018.395,175.250,377.943,167.710,52.050,159.692
C05146=1018.390,175.001,377.965,167.706,52.059,159.693
C05147=1018.385,174.752,377.986,167.702,52.067,159.694
C05148=1018.380,174.503,378.007,167.699,52.075,159.695
C05149=1018.375,174.253,378.029,167.695,52.084,159.696
C05150=1018.369,174.005,378.050,167.690,52.092,159.696
C05151=1018.365,173.755,378.071,167.687,52.101,159.698
C05152=1018.360,173.506,378.093,167.683,52.109,159.699
C05153=1018.354,173.258,378.115,167.679,52.118,159.700
C05154=1018.350,173.008,378.136,167.675,52.126,159.700
C05155=1018.344,172.760,378.157,167.672,52.135,159.702
C05156=1018.340,172.510,378.178,167.668,52.143,159.703
C05157=1018.335,172.262,378.200,167.664,52.152,159.704
C05158=1018.330,172.013,378.220,167.660,52.160,159.704
C05159=1018.325,171.764,378.242,167.656,52.168,159.705
C05160=1018.320,171.482,378.266,167.652,52.178,159.707
C05161=1018.314,171.200,378.290,167.648,52.188,159.708
C05162=1018.308,170.920,378.314,167.644,52.197,159.709
C05163=1018.303,170.638,378.338,167.639,52.207,159.710
C05164=1018.297,170.390,378.359,167.635,52.215,159.711
C05165=1018.293,170.141,378.380,167.632,52.224,159.712
C05166=1018.288,169.892,378.402,167.628,52.232,159.713
C05167=1018.283,169.643,378.423,167.624,52.240,159.714
C05168=1018.278,169.393,378.444,167.620,52.249,159.715
C05169=1018.273,169.145,378.465,167.616,52.257,159.716
C05170=1018.268,168.895,378.486,167.613,52.266,159.717
C05171=1018.263,168.646,378.508,167.609,52.274,159.718
C05172=1018.258,168.397,378.529,167.606,52.283,159.719
C05173=1018.254,168.148,378.550,167.601,52.291,159.720
C05174=1018.248,167.899,378.571,167.598,52.300,159.721
C05175=1018.244,167.650,378.592,167.594,52.308,159.722
C05176=1018.239,167.400,378.613,167.590,52.316,159.723
C05177=1018.233,167.152,378.635,167.587,52.325,159.724
C05178=1018.229,166.903,378.656,167.583,52.333,159.725
C05179=1018.224,166.653,378.676,167.580,52.342,159.726
C05180=1018.219,166.405,378.698,167.575,52.350,159.727
C05181=1018.214,166.155,378.719,167.572,52.359,159.728
C05182=1018.209,165.906,378.740,167.568,52.367,159.729
C05183=1018.205,165.658,378.761,167.565,52.375,159.730
C05184=1018.200,165.409,378.782,167.561,52.384,159.731
C05185=1018.195,165.159,378.803,167.558,52.392,159.732
C05186=1018.191,164.910,378.824,167.554,52.401,159.733
C05187=1018.185,164.661,378.846,167.551,52.409,159.734
C05188=1018.180,164.412,378.867,167.547,52.418,159.735
C05189=1018.176,164.163,378.888,167.543,52.426,159.736
C05190=1018.171,163.913,378.908,167.539,52.434,159.737
C05191=1018.167,163.665,378.930,167.536,52.443,159.738
C05192=1018.161,163.416,378.950,167.532,52.451,159.739
C05193=1018.157,163.167,378.972,167.529,52.460,159.740
C05194=1018.152,162.917,378.993,167.525,52.468,159.741
C05195=1018.147,162.668,379.013,167.521,52.476,159.742
C05196=1018.142,162.419,379.035,167.518,52.485,159.743
C05197=1018.137,162.171,379.055,167.514,52.493,159.744
C05198=1018.133,161.922,379.077,167.511,52.502,159.745
C05199=1018.128,161.672,379.098,167.507,52.510,159.746
C05200=1018.123,161.423,379.118,167.504,52.518,159.747
C05201=1018.119,161.174,379.139,167.500,52.527,159.748
C05202=1018.114,160.925,379.160,167.497,52.535,159.749
C05203=1018.109,160.676,379.181,167.493,52.544,159.750
C05204=1018.104,160.427,379.202,167.490,52.552,159.751
C05205=1018.099,160.178,379.223,167.486,52.560,159.752
C05206=1018.096,159.929,379.244,167.483,52.569,159.753
C05207=1018.090,159.680,379.264,167.479,52.577,159.754
C05208=1018.086,159.430,379.286,167.476,52.586,159.755
C05209=1018.080,159.181,379.306,167.472,52.594,159.756
C05210=1018.077,158.933,379.327,167.468,52.602,159.757
C05211=1018.072,158.683,379.348,167.465,52.611,159.758
C05212=1018.067,158.434,379.369,167.461,52.620,159.759
C05213=1018.062,158.185,379.389,167.457,52.629,159.760
C05214=1018.056,157.936,379.410,167.454,52.637,159.761
C05215=1018.052,157.687,379.430,167.450,52.645,159.762
C05216=1018.047,157.438,379.450,167.447,52.654,159.763
C05217=1018.042,157.188,379.471,167.443,52.662,159.764
C05218=1018.037,156.939,379.492,167.440,52.671,159.765
C05219=1018.032,156.691,379.512,167.436,52.681,159.766
C05220=1018.027,156.441,379.532,167.432,52.689,159.767
C05221=1018.022,156.192,379.552,167.429,52.698,159.768
C05222=1018.017,155.943,379.573,167.426,52.706,159.769
C05223=1018.012,155.694,379.593,167.422,52.715,159.770
C05224=1018.007,155.412,379.616,167.418,52.724,159.772
C05225=1018.001,155.131,379.639,167.415,52.734,159.773
C05226=1017.995,154.849,379.663,167.410,52.744,159.774
C05227=1017.990,154.568,379.685,167.407,52.754,159.775
C05228=1017.985,154.319,379.705,167.403,52.762,159.776
C05229=1017.980,154.070,379.725,167.400,52.771,159.777
C05230=1017.975,153.820,379.746,167.397,52.779,159.778
C05231=1017.971,153.572,379.766,167.393,52.788,159.779
C05232=1017.966,153.322,379.786,167.390,52.796,159.780
C05233=1017.961,153.073,379.807,167.386,52.805,159.781
C05234=1017.956,152.824,379.827,167.382,52.814,159.782
C05235=1017.951,152.575,379.847,167.379,52.823,159.783
C05236=1017.946,152.326,379.867,167.375,52.832,159.784
C05237=1017.941,152.076,379.888,167.372,52.840,159.785
C05238=1017.936,151.827,379.907,167.369,52.849,159.787
C05239=1017.931,151.578,379.928,167.365,52.858,159.788
C05240=1017.926,151.328,379.948,167.362,52.866,159.789
C05241=1017.921,151.080,379.968,167.359,52.875,159.790
C05242=1017.917,150.830,379.988,167.355,52.883,159.791
C05243=1017.912,150.582,380.008,167.352,52.892,159.792
C05244=1017.907,150.332,380.028,167.349,52.901,159.793
C05245=1017.902,150.083,380.048,167.345,52.909,159.794
C05246=1017.897,149.834,380.068,167.341,52.918,159.795
C05247=1017.891,149.585,380.088,167.338,52.927,159.796
C05248=1017.886,149.335,380.108,167.334,52.936,159.797
C05249=1017.882,149.087,380.128,167.331,52.944,159.798
C05250=1017.877,148.837,380.148,167.328,52.953,159.799
C05251=1017.872,148.589,380.168,167.324,52.962,159.800
C05252=1017.867,148.339,380.188,167.321,52.970,159.801
C05253=1017.862,148.091,380.208,167.318,52.979,159.802
C05254=1017.858,147.841,380.228,167.314,52.988,159.804
C05255=1017.852,147.592,380.248,167.311,52.996,159.805
C05256=1017.848,147.343,380.268,167.308,53.005,159.806
C05257=1017.843,147.093,380.288,167.305,53.014,159.807
C05258=1017.838,146.845,380.308,167.301,53.022,159.808
C05259=1017.833,146.595,380.328,167.298,53.031,159.809
C05260=1017.828,146.347,380.347,167.295,53.040,159.810
C05261=1017.823,146.097,380.367,167.291,53.048,159.811
C05262=1017.818,145.847,380.387,167.288,53.057,159.812
C05263=1017.813,145.599,380.407,167.285,53.066,159.813
C05264=1017.808,145.349,380.427,167.281,53.074,159.814
C05265=1017.803,145.100,380.446,167.278,53.083,159.815
C05266=1017.798,144.851,380.466,167.275,53.092,159.817
C05267=1017.794,144.602,380.486,167.271,53.101,159.818
C05268=1017.789,144.352,380.506,167.268,53.110,159.819
C05269=1017.784,144.104,380.525,167.264,53.118,159.820
C05270=1017.779,143.854,380.544,167.261,53.127,159.821
C05271=1017.774,143.606,380.565,167.258,53.136,159.822
C05272=1017.768,143.356,380.584,167.255,53.145,159.823
C05273=1017.764,143.107,380.603,167.251,53.153,159.824
C05274=1017.759,142.857,380.623,167.248,53.162,159.825
C05275=1017.754,142.609,380.642,167.245,53.171,159.826
C05276=1017.749,142.359,380.663,167.242,53.180,159.827
C05277=1017.744,142.110,380.682,167.238,53.188,159.828
C05278=1017.739,141.861,380.701,167.235,53.197,159.829
C05279=1017.734,141.612,380.721,167.232,53.206,159.831
C05280=1017.729,141.362,380.741,167.228,53.214,159.832
C05281=1017.724,141.114,380.759,167.225,53.223,159.833
C05282=1017.719,140.864,380.779,167.222,53.232,159.834
C05283=1017.715,140.615,380.799,167.219,53.241,159.835
C05284=1017.709,140.366,380.819,167.215,53.249,159.836
C05285=1017.705,140.117,380.838,167.212,53.258,159.837
C05286=1017.700,139.867,380.858,167.209,53.267,159.838
C05287=1017.695,139.618,380.877,167.206,53.276,159.839
C05288=1017.689,139.337,380.899,167.202,53.286,159.840
C05289=1017.684,139.055,380.921,167.198,53.296,159.842
C05290=1017.679,138.774,380.943,167.195,53.306,159.843
C05291=1017.673,138.492,380.965,167.191,53.316,159.844
C05292=1017.668,138.242,380.985,167.188,53.325,159.845
C05293=1017.664,137.993,381.004,167.184,53.333,159.846
C05294=1017.658,137.744,381.024,167.181,53.342,159.847
C05295=1017.654,137.495,381.043,167.178,53.351,159.849
C05296=1017.649,137.246,381.062,167.175,53.360,159.850
C05297=1017.644,136.996,381.082,167.171,53.368,159.851
C05298=1017.639,136.748,381.101,167.168,53.377,159.852
C05299=1017.634,136.498,381.121,167.165,53.386,159.853
C05300=1017.629,136.249,381.139,167.162,53.395,159.854
C05301=1017.624,136.000,381.159,167.159,53.403,159.855
C05302=1017.618,135.751,381.178,167.156,53.412,159.856
C05303=1017.614,135.501,381.197,167.153,53.421,159.857
C05304=1017.609,135.252,381.216,167.149,53.430,159.859
C05305=1017.604,135.003,381.236,167.146,53.439,159.860
C05306=1017.599,134.754,381.254,167.143,53.447,159.861
C05307=1017.594,134.504,381.274,167.140,53.456,159.862
C05308=1017.589,134.255,381.293,167.137,53.465,159.863
C05309=1017.584,134.006,381.311,167.134,53.474,159.864
C05310=1017.580,133.756,381.331,167.131,53.483,159.865
C05311=1017.574,133.507,381.350,167.127,53.492,159.866
C05312=1017.569,133.259,381.369,167.124,53.501,159.867
C05313=1017.564,133.009,381.389,167.121,53.510,159.868
C05314=1017.560,132.760,381.407,167.118,53.519,159.870
C05315=1017.555,132.511,381.426,167.114,53.527,159.871
C05316=1017.550,132.261,381.446,167.111,53.536,159.872
C05317=1017.545,132.012,381.465,167.108,53.545,159.873
C05318=1017.540,131.763,381.484,167.105,53.554,159.874
C05319=1017.535,131.513,381.503,167.102,53.563,159.875
C05320=1017.530,131.264,381.522,167.099,53.571,159.876
C05321=1017.525,131.016,381.541,167.096,53.580,159.877
C05322=1017.520,130.767,381.560,167.093,53.589,159.878
C05323=1017.516,130.516,381.579,167.090,53.598,159.880
C05324=1017.511,130.268,381.598,167.086,53.607,159.881
C05325=1017.506,130.019,381.617,167.083,53.616,159.882
C05326=1017.501,129.769,381.636,167.081,53.624,159.883
C05327=1017.496,129.520,381.655,167.078,53.633,159.884
C05328=1017.492,129.270,381.673,167.074,53.643,159.885
C05329=1017.486,129.021,381.693,167.071,53.652,159.886
C05330=1017.481,128.771,381.711,167.068,53.660,159.887
C05331=1017.476,128.523,381.730,167.065,53.669,159.888
C05332=1017.471,128.273,381.748,167.061,53.678,159.890
C05333=1017.466,128.024,381.767,167.058,53.687,159.891
C05334=1017.461,127.775,381.785,167.055,53.696,159.892
C05335=1017.456,127.526,381.804,167.052,53.705,159.893
C05336=1017.450,127.276,381.823,167.049,53.714,159.894
C05337=1017.445,127.027,381.842,167.046,53.723,159.895
C05338=1017.441,126.778,381.860,167.043,53.732,159.897
C05339=1017.435,126.529,381.879,167.040,53.741,159.898
C05340=1017.430,126.279,381.897,167.037,53.750,159.899
C05341=1017.425,126.030,381.916,167.034,53.759,159.900
C05342=1017.420,125.781,381.934,167.031,53.767,159.901
C05343=1017.415,125.532,381.953,167.028,53.777,159.902
C05344=1017.410,125.282,381.972,167.025,53.786,159.903
C05345=1017.405,125.033,381.990,167.022,53.795,159.904
C05346=1017.400,124.784,382.009,167.019,53.804,159.906
C05347=1017.396,124.534,382.027,167.016,53.813,159.907
C05348=1017.391,124.286,382.046,167.013,53.822,159.908
C05349=1017.385,124.036,382.065,167.010,53.831,159.909
C05350=1017.380,123.787,382.084,167.007,53.840,159.910
C05351=1017.375,123.537,382.102,167.004,53.848,159.911
C05352=1017.369,123.256,382.123,167.000,53.858,159.913
C05353=1017.364,122.974,382.143,166.997,53.868,159.914
C05354=1017.358,122.692,382.164,166.993,53.879,159.915
C05355=1017.353,122.411,382.186,166.989,53.889,159.916
C05356=1017.348,122.162,382.204,166.987,53.898,159.917
C05357=1017.344,121.912,382.222,166.984,53.907,159.919
C05358=1017.338,121.663,382.241,166.981,53.916,159.920
C05359=1017.333,121.413,382.259,166.979,53.925,159.921
C05360=1017.328,121.164,382.277,166.976,53.934,159.922
C05361=1017.323,120.915,382.296,166.972,53.942,159.923
C05362=1017.318,120.666,382.315,166.969,53.951,159.924
C05363=1017.314,120.417,382.333,166.966,53.960,159.926
C05364=1017.309,120.168,382.352,166.963,53.969,159.927
C05365=1017.303,119.918,382.370,166.960,53.978,159.928
C05366=1017.298,119.669,382.388,166.957,53.987,159.929
C05367=1017.293,119.420,382.407,166.954,53.996,159.930
C05368=1017.288,119.170,382.425,166.951,54.005,159.931
C05369=1017.284,118.921,382.443,166.948,54.014,159.932
C05370=1017.279,118.672,382.462,166.945,54.023,159.934
C05371=1017.274,118.423,382.480,166.942,54.031,159.934
C05372=1017.269,118.174,382.499,166.939,54.040,159.936
C05373=1017.264,117.924,382.517,166.937,54.049,159.937
C05374=1017.260,117.675,382.535,166.934,54.058,159.938
C05375=1017.254,117.426,382.554,166.931,54.067,159.939
C05376=1017.249,117.176,382.572,166.928,54.076,159.940
C05377=1017.244,116.927,382.591,166.925,54.085,159.941
C05378=1017.240,116.677,382.609,166.922,54.094,159.943
C05379=1017.235,116.428,382.627,166.919,54.103,159.944
C05380=1017.230,116.179,382.646,166.916,54.111,159.945
C05381=1017.226,115.930,382.665,166.913,54.120,159.946
C05382=1017.221,115.680,382.683,166.911,54.129,159.947
C05383=1017.216,115.431,382.701,166.907,54.137,159.948
C05384=1017.211,115.182,382.719,166.904,54.147,159.949
C05385=1017.206,114.933,382.738,166.902,54.156,159.950
C05386=1017.201,114.684,382.756,166.899,54.165,159.952
C05387=1017.197,114.434,382.774,166.895,54.173,159.953
C05388=1017.192,114.185,382.792,166.892,54.182,159.954
C05389=1017.187,113.936,382.811,166.890,54.191,159.955
C05390=1017.182,113.686,382.829,166.887,54.199,159.956
C05391=1017.177,113.437,382.847,166.884,54.208,159.957
C05392=1017.172,113.188,382.866,166.881,54.218,159.958
C05393=1017.168,112.939,382.884,166.878,54.227,159.960
C05394=1017.163,112.689,382.902,166.875,54.235,159.960
C05395=1017.158,112.440,382.920,166.873,54.244,159.962
C05396=1017.153,112.191,382.938,166.870,54.253,159.963
C05397=1017.148,111.941,382.957,166.867,54.261,159.964
C05398=1017.144,111.692,382.975,166.864,54.270,159.965
C05399=1017.138,111.443,382.992,166.861,54.280,159.966
C05400=1017.133,111.194,383.010,166.858,54.289,159.967
C05401=1017.129,110.944,383.029,166.855,54.298,159.969
C05402=1017.124,110.695,383.047,166.852,54.307,159.970
C05403=1017.118,110.446,383.064,166.849,54.315,159.971
C05404=1017.114,110.196,383.082,166.846,54.324,159.972
C05405=1017.109,109.947,383.100,166.843,54.334,159.973
C05406=1017.104,109.698,383.117,166.842,54.342,159.974
C05407=1017.099,109.448,383.136,166.839,54.351,159.976
C05408=1017.094,109.199,383.154,166.835,54.360,159.977
C05409=1017.088,108.950,383.171,166.832,54.369,159.978
C05410=1017.084,108.700,383.190,166.830,54.378,159.979
C05411=1017.079,108.450,383.207,166.827,54.387,159.980
C05412=1017.074,108.201,383.225,166.824,54.396,159.981
C05413=1017.069,107.952,383.243,166.821,54.406,159.982
C05414=1017.063,107.703,383.260,166.818,54.415,159.984
C05415=1017.059,107.453,383.278,166.815,54.424,159.985
C05416=1017.053,107.172,383.298,166.812,54.434,159.986
C05417=1017.047,106.890,383.318,166.808,54.444,159.987
C05418=1017.042,106.608,383.338,166.805,54.455,159.989
C05419=1017.035,106.327,383.358,166.803,54.464,159.990
C05420=1017.032,106.078,383.375,166.800,54.474,159.991
C05421=1017.026,105.829,383.393,166.797,54.483,159.993
C05422=1017.021,105.579,383.411,166.794,54.491,159.993
C05423=1017.016,105.330,383.428,166.791,54.500,159.995
C05424=1017.011,105.080,383.446,166.788,54.509,159.996
C05425=1017.006,104.831,383.463,166.785,54.519,159.997
C05426=1017.001,104.582,383.482,166.782,54.528,159.998
C05427=1016.997,104.332,383.499,166.780,54.537,159.999
C05428=1016.991,104.083,383.517,166.776,54.545,160.000
C05429=1016.986,103.833,383.535,166.773,54.555,160.002
C05430=1016.982,103.585,383.551,166.772,54.563,160.003
C05431=1016.977,103.335,383.569,166.769,54.573,160.004
C05432=1016.971,103.086,383.587,166.766,54.582,160.005
C05433=1016.967,102.836,383.604,166.763,54.591,160.006
C05434=1016.961,102.587,383.622,166.760,54.599,160.007
C05435=1016.957,102.338,383.640,166.757,54.608,160.009
C05436=1016.951,102.088,383.657,166.754,54.618,160.010
C05437=1016.947,101.839,383.675,166.751,54.627,160.011
C05438=1016.942,101.590,383.692,166.749,54.635,160.012
C05439=1016.937,101.340,383.710,166.746,54.644,160.013
C05440=1016.932,101.091,383.728,166.744,54.653,160.014
C05441=1016.927,100.841,383.745,166.741,54.662,160.016
C05442=1016.922,100.592,383.763,166.738,54.672,160.017
C05443=1016.917,100.343,383.780,166.735,54.680,160.018
C05444=1016.913,100.094,383.798,166.732,54.689,160.019
C05445=1016.907,99.845,383.815,166.730,54.698,160.020
C05446=1016.903,99.595,383.833,166.727,54.707,160.021
C05447=1016.897,99.346,383.850,166.724,54.716,160.022
C05448=1016.893,99.096,383.868,166.721,54.725,160.024
C05449=1016.887,98.847,383.885,166.718,54.734,160.025
C05450=1016.883,98.598,383.902,166.716,54.743,160.026
C05451=1016.878,98.348,383.920,166.713,54.752,160.027
C05452=1016.873,98.099,383.937,166.710,54.761,160.028
C05453=1016.868,97.849,383.954,166.707,54.770,160.029
C05454=1016.862,97.600,383.971,166.704,54.779,160.031
C05455=1016.858,97.351,383.988,166.701,54.789,160.032
C05456=1016.853,97.102,384.006,166.700,54.797,160.033
